		/////////////////////////////////
		E_CRYO_CTRL_STATE.WARMING_UP:
		/////////////////////////////////
		//
		// Trigger temperature ramp to in_ptr_Cryo_Ctrl^.cfg.lrTemp_Warm (~10C)
		SIM_Temp_Mirror.M_RampTo(
			in_lrValueEnd	:= in_ptr_Cryo_Ctrl^.cfg.lrTemp_Warm + 1.0,
			in_nPeriod		:= nRampPeriod);
			
			
		// Trigger temperature ramp to in_ptr_Cryo_Ctrl^.cfg.lrTemp_Warm (~10C)
		// Speed up the ramp compared to the Bench, so
		// DET temperature is slightly higher during warm-up.
		// The final temperature is the same as for the Bench.
		SIM_Temp_DET.M_RampTo(
			in_lrValueEnd	:= in_ptr_Cryo_Ctrl^.cfg.lrTemp_Warm + 1.0,
			in_nPeriod		:= nRampPeriod - 2000);
			
		/////////////////////////////////
		E_CRYO_CTRL_STATE.REPRESSURIZING:
		/////////////////////////////////
		//
		// Trigger Cryo vacuum ramp to atmospheric pressure ~820 mbar
		SIM_Pressure_Cryo.M_RampTo(
			in_lrValueEnd	:= 820.0,
			in_nPeriod		:= 17000);
			
		// Follow the same ramp with Evac but a bit slower.
		SIM_Pressure_Evac.M_RampTo(
			in_lrValueEnd	:= 820.0,
			in_nPeriod		:= 20000);
	END_CASE

END_IF


//
// Evacuation Pressure simulation
//
// Capture Evacuation ON/OFF trigger
trgEvacOn(CLK := in_ptr_Cryo_Ctrl^.ctrl.bEnable_Evac);
trgEvacOff(CLK := in_ptr_Cryo_Ctrl^.ctrl.bEnable_Evac);
IF	trgEvacOn.Q THEN
	// Trigger vacuum ramp 0.0001 mbar below Good Vacuum
	SIM_Pressure_Cryo.M_StartCurve(
		in_lrValueEnd	:= in_ptr_Cryo_Ctrl^.Pressure_Cryo.in_lrLimitGoodVac - 0.0001, 
		in_nPeriod		:= 20000, 
		in_lrCurveScale	:= 0.3);
ELSIF trgEvacOff.Q THEN
	// Evacuation stopped.
	// Keep the pressure as it is.
	SIM_Pressure_Cryo.M_Stop();
END_IF


//
// If Turbo Pump is running, keep Evacuation pressure 1.0e-05 below the Cryo pressure.
// Value is calculated on every cycle.
//
IF in_ptr_Cryo_Ctrl^.EvacSys.stat.bTurboPumpON THEN
	SIM_Pressure_Evac.M_SetValue(SIM_Pressure_Cryo.lrPress - 1.0E-05);
END_IF


//
// To get more realistic evacuation,
// Restart simulated curve when inVacuum is triggered.
//
//trgInVacuum(CLK := in_ptr_Cryo_Ctrl^.Pressure_Cryo.stat.bInVacuum);
trgInVacuum(CLK := in_ptr_Cryo_Ctrl^.stat.bInVacuum);
IF trgInVacuum.Q THEN
	SIM_Pressure_Cryo.M_StartCurve(
		in_lrValueEnd	:= in_ptr_Cryo_Ctrl^.Pressure_Cryo.in_lrLimitGoodVac - 0.0001, 
		in_nPeriod		:= 10000, 
		in_lrCurveScale	:= 0.3);
END_IF

			
//
// Capture events when buttons are released 
// and temperature transitions interrupted.
//

// Capture pre-cooling, cooling or warmup button release.
// Stop ramping in that case.
trgPrecoolOff	(CLK:=in_ptr_Cryo_Ctrl^.ctrl.bEnable_Precool);
trgCoolOff		(CLK:=in_ptr_Cryo_Ctrl^.ctrl.bEnable_Cool);
trgWarmupOff	(CLK:=in_ptr_Cryo_Ctrl^.ctrl.bEnable_Warmup);

IF	trgPrecoolOff.Q OR trgCoolOff.Q OR trgWarmupOff.Q	THEN
	SIM_Temp_Mirror.M_Stop();
	SIM_Temp_DET.M_Stop();
END_IF

END_FUNCTION_BLOCK

// POUs/System/FB_CRYO_CTRL
// Cryogenic Controller Example - ESO IRATEC
FUNCTION_BLOCK FB_CRYO_CTRL
VAR_INPUT
END_VAR
VAR

	///////////////////////////
	// Configuration parameters
	///////////////////////////
	cfg:	T_CRYO_CFG;
	
	/////////////////////
	// Control parameters
	/////////////////////
	ctrl:	T_CRYO_CTRL;

	/////////////////////
	// Status parameters
	/////////////////////
	stat:	T_CRYO_STAT;


	/////////////////////
	// System Logging
	/////////////////////
	syslog:	T_CRYO_LOG;


	/////////////////////
	// Local variables
	/////////////////////



	{attribute 'OPC.UA.DA' := '0'}
	timer:		TON;		// Timer for commands
	
	{attribute 'OPC.UA.DA' := '0'}
	ptrLog:		ARRAY [0..9] OF POINTER TO STRING(80);
	{attribute 'OPC.UA.DA' := '0'}
	nLogPos:	INT := -1;
	
	

//////////////////////////////////////////////
//             Controllers
//////////////////////////////////////////////

//
// LN2 Valve control
//
	{attribute 'OPC.UA.DA' := '1'}
	LN2: 			FB_CRYO_LN2_CTRL;
	
//
// Repressurizing Valve control
//
	{attribute 'OPC.UA.DA' := '1'}
	RepressValve:	FB_CRYO_VALVE_CTRL;
	
	
//
// Evacuation Valve control
//
	EvacSys:	FB_CRYO_EVACUATION_SYSTEM;

//
// Heater control
//
	{attribute 'OPC.UA.DA' := '1'}
	Heater: 		FB_CRYO_HEATER_CTRL;
	
//
// CCC control
//
	{attribute 'OPC.UA.DA' := '1'}
	CCC:			FB_CRYO_CCC_CTRL;

//
// CCC control
//
//	{attribute 'OPC.UA.DA' := '1'}
	Lakeshore:		FB_LAKESHORE_RS;
	
	// Compressor	
	cpa:	FB_CRYO_CPA;

//////////////////////////////////////////////
//             Sensors
//////////////////////////////////////////////
 
//
// VACUUM Sensors
//
	{attribute 'OPC.UA.DA' := '1'}
	Pressure_Cryo:		FB_CRYO_PRESSURE;	
	{attribute 'OPC.UA.DA' := '1'}
	Pressure_Evac:		FB_CRYO_PRESSURE;	
	
 
///////////////////////////////////////////////////////
//                  Temperatures
///////////////////////////////////////////////////////
 
//
// PT100 Temperatures
//
	Temp_Ambient:		FB_CRYO_TEMPERATURE;	// Ambient temperature
	Temp_ColdBench:		FB_CRYO_TEMPERATURE;	// Cold Bench temperature
	Temp_LN2_Exhaust:	FB_CRYO_TEMPERATURE;	// LN2 Exhaust temperature
	Temp_LN2_Inlet:		FB_CRYO_TEMPERATURE;	// LN2 Inlet   temperature
	Temp_Mirror:		FB_CRYO_TEMPERATURE;	// Entrance Mirror temperature
	Temp_WarmUp:		FB_CRYO_TEMPERATURE;	// Reference temperature for WarmUp

//
// Lakeshore temperatures
//
	Temp_DET:			FB_CRYO_TEMPERATURE;	// Lakeshore Channel A
	Temp_HeatShield:	FB_CRYO_TEMPERATURE;	// Heat Shield Lakeshore Channel B
 
//
// IRATEC specific Temperatures
//
	Temp_FW:			FB_CRYO_TEMPERATURE;	// Filter Wheel temperature

	

//
// System triggers
//	
	{attribute 'OPC.UA.DA' := '0'}
	trgPrecool:			R_TRIG;
	{attribute 'OPC.UA.DA' := '0'}
	trgCool:			R_TRIG;
	{attribute 'OPC.UA.DA' := '0'}
	trgWarmup:			R_TRIG;
	{attribute 'OPC.UA.DA' := '0'}
	trgRepress:			R_TRIG;
	{attribute 'OPC.UA.DA' := '0'}
	trgEvacOn:			R_TRIG;
	{attribute 'OPC.UA.DA' := '0'}
	trgEvacOff:			F_TRIG;

//
//	Input signals
//	
	i_bEvacRootPumpOK		AT%I*:	BOOL;
	i_bEvacTurboPumpOK		AT%I*:	BOOL;
	i_bEmergencySTOP		AT%I*:	BOOL;
	i_bManualOverride		AT%I*:	BOOL;
	i_bVacPumpConnected		AT%I*:	BOOL;
	i_bLN2TankConnected		AT%I*:	BOOL;
	i_bRepressLN2Connected	AT%I*:	BOOL;


//
// Dummy values for simulation, etc.
//
	// Dummy OP state for mapping of simulated devices.
	q_nStateDummy	AT%Q*:	UINT := 8;		

	
END_VAR

// Increment cycle counter
stat.nCycleCounter := stat.nCycleCounter + 1;

// Wait until the controller is configured.
IF NOT stat.bConfigured THEN
	M_Configure(); 
	RETURN;
END_IF


//
// Read Temperature and Pressure Sensors
//
M_ReadSensors();


//
// Check for sensor HW errors
//
M_CheckForSensorErrors();



///////////////////
// System Operation
///////////////////

//
// Execute Controllers
//
M_ExecuteControllers();


//
// Capture system commands
//
M_CheckForCommands();


//
// Perform a safety check
//
M_SafetyCheck();


//
// Execute system state machine
//
M_StateMachine();

METHOD M_CheckForCommands
VAR_INPUT
END_VAR
// Capture precooling command
trgPrecool(CLK := ctrl.bEnable_Precool);
IF	trgPrecool.Q AND 
	(stat.nState = E_CRYO_CTRL_STATE.WARM_VACUUM OR stat.nState = E_CRYO_CTRL_STATE.PRE_COOLED) THEN
	ctrl.bExecute	:= TRUE;
	ctrl.nCommand	:= E_CRYO_CTRL_CMD.PRECOOL;
END_IF


// Capture Cool command
trgCool(CLK := ctrl.bEnable_Cool);
IF	trgCool.Q AND stat.nState = E_CRYO_CTRL_STATE.PRE_COOLED THEN
	ctrl.bExecute	:= TRUE;
	ctrl.nCommand	:= E_CRYO_CTRL_CMD.COOL;
END_IF


// Capture Warmup command
trgWarmup(CLK := ctrl.bEnable_Warmup);
IF	trgWarmup.Q AND 
	(stat.nState = E_CRYO_CTRL_STATE.PRE_COOLED OR stat.nState = E_CRYO_CTRL_STATE.COLD) THEN
	ctrl.bExecute	:= TRUE;
	ctrl.nCommand	:= E_CRYO_CTRL_CMD.WARM_UP;
END_IF


// Capture Repressure command
trgRepress(CLK := ctrl.bEnable_RepressCtrl);
IF	trgRepress.Q AND 
	(stat.nState = E_CRYO_CTRL_STATE.WARM_VACUUM) THEN
	ctrl.bExecute	:= TRUE;
	ctrl.nCommand	:= E_CRYO_CTRL_CMD.REPRESSURIZE;
END_IF


// Capture Evacuation ON/OFF trigger
trgEvacOn(CLK := ctrl.bEnable_Evac);
trgEvacOff(CLK := ctrl.bEnable_Evac);
IF	trgEvacOn.Q AND NOT ctrl.bEnable_RepressSys THEN
	ctrl.bEnable_Evac	:= TRUE;
	M_SysLog('Evacuation started.');
ELSIF trgEvacOff.Q THEN
	ctrl.bEnable_Evac	:= FALSE;
	M_SysLog('Evacuation stopped.');
END_IF
END_METHOD

METHOD M_CheckForSensorErrors
VAR_INPUT
END_VAR
////////////////////////////////////////////////
// Check for errors by testing the 'Valid' flag.
////////////////////////////////////////////////
IF		NOT Pressure_Cryo.stat.bValid	THEN
	stat.bError	:= TRUE;
	stat.sState	:= 'Cryo Vacuum gauge problem';
	stat.nState	:= E_CRYO_CTRL_STATE.ERROR;
ELSIF	NOT Temp_Mirror.stat.bValid	THEN
	stat.bError	:= TRUE;
	stat.sState	:= 'Mirror Temperature sensor problem';
	stat.nState	:= E_CRYO_CTRL_STATE.ERROR;
ELSE
	stat.bError	:= FALSE;
	stat.sState	:= '';
END_IF


///////////////////////
// Check for Interlocks
///////////////////////

//
// Evacuation and Repressurization are mutually exclusive.
//
IF EvacSys.in_bEnable THEN
	ctrl.bEnable_RepressSys	:= FALSE;
ELSIF RepressValve.in_bEnable THEN
	ctrl.bEnable_Evac	:= FALSE;
END_IF

//
// Disable control in failure state
//
IF stat.bError THEN
	ctrl.bEnable_Precool	:= FALSE;
	ctrl.bEnable_Cool 		:= FALSE;
	ctrl.bEnable_Warmup		:= FALSE;
END_IF
END_METHOD

METHOD M_CheckLakeshoreCommand
VAR_INPUT
END_VAR
(* TODO

IF ctrl.bLS_UpdateSETP THEN
	// Reset trigger flag
	ctrl.bLS_UpdateSETP	:= FALSE;
	
	// Safety
	IF ctrl.lrLS_RAMP > 1.0 THEN
		ctrl.lrLS_RAMP	:= 1.0;
	ELSIF ctrl.lrLS_RAMP < 0.0 THEN
		ctrl.lrLS_RAMP	:= 0.0;
	END_IF
	
	// Set the mode
	IF ctrl.nLS_Mode <> E_CRYO_LAKESHORE_MODE.MONITORING THEN
		Lakeshore.M_SetMode(ctrl.nLS_Mode);
	ELSE
		RETURN;	// Nothing to do
	END_IF
ELSE
	RETURN;	// Nothing to do
END_IF




CASE ctrl.nLS_Mode OF
	E_CRYO_LAKESHORE_MODE.MONITORING,
	E_CRYO_LAKESHORE_MODE.COOLING,
	E_CRYO_LAKESHORE_MODE.WARMUP,
	E_CRYO_LAKESHORE_MODE.COOLING_UPDATE,
	E_CRYO_LAKESHORE_MODE.WARMUP_UPDATE:
		Lakeshore.M_SetMode(E_CRYO_LAKESHORE_MODE.MONITORING);	// No action
		
	E_CRYO_LAKESHORE_MODE.SINGLE_SETUP:
		IF stat.nState = E_CRYO_CTRL_STATE.COLD THEN
			Lakeshore.M_SetParams(
				in_nPID_A_P			:= cfg.LS_W_PID_A_P, 
				in_nPID_A_I			:= cfg.LS_W_PID_A_I, 
				in_nPID_A_D			:= cfg.LS_W_PID_A_D, 
				in_nHeater_Range	:= cfg.LS_W_Heater_Range, 
				in_lrCtrlRamp		:= ctrl.lrLS_RAMP, 
				in_lrSetpoint_A		:= ctrl.lrLS_SETP);
		END_IF
	ELSE
		Lakeshore.M_SetMode(E_CRYO_LAKESHORE_MODE.MONITORING);	// No action
END_CASE
*)
END_METHOD

// Method to check status of the cryostat vacuum.
// TODO: The limits might depend on the temperature.
METHOD M_CheckVacuum
VAR_INPUT
END_VAR
IF Pressure_Cryo.stat.bValid  THEN
	IF Pressure_Cryo.stat.lrPressure < cfg.lrPress_GoodVac THEN
		stat.bInVacuum	:= TRUE;
		stat.bGoodVacuum:= TRUE;
	ELSIF Pressure_Cryo.stat.lrPressure < cfg.lrPress_InVac THEN
		stat.bInVacuum	:= TRUE;
		stat.bGoodVacuum:= FALSE;
	ELSE
		stat.bInVacuum	:= FALSE;
		stat.bGoodVacuum:= FALSE;
	END_IF 
ELSE
	stat.bInVacuum	:= FALSE;
	stat.bGoodVacuum:= FALSE;
END_IF
END_METHOD

METHOD M_Configure
VAR_INPUT
END_VAR
IF stat.bConfigured THEN
	RETURN;
ELSIF stat.nCycleCounter = 100 THEN
	// Set pointers to system logs.
	ptrLog[0] := ADR(syslog.s0);
	ptrLog[1] := ADR(syslog.s1);
	ptrLog[2] := ADR(syslog.s2);
	ptrLog[3] := ADR(syslog.s3);
	ptrLog[4] := ADR(syslog.s4);
	ptrLog[5] := ADR(syslog.s5);
	ptrLog[6] := ADR(syslog.s6);
	ptrLog[7] := ADR(syslog.s7);
	ptrLog[8] := ADR(syslog.s8);
	ptrLog[9] := ADR(syslog.s9);
ELSIF stat.nCycleCounter > 200 THEN
	stat.bConfigured	:= TRUE;
ELSE
	RETURN;
END_IF
END_METHOD

METHOD M_ExecuteControllers
VAR
END_VAR
//
// Controllers, i.e. LN2 cooler, Heater, ...
//

// Activate Lakeshore SETP command, if any (see ctrl.xxLS_...)
M_CheckLakeshoreCommand();

// Execute Lakeshore 340 controller
Lakeshore(
	in_bSimulation	:= TRUE,
	in_sName		:= 'LS340',
	in_nModel		:= 340, 
	in_bAutoMonitor	:= TRUE, 
	in_nPeriod 		:= 2000,
	in_sCmdSuffix	:= '$0D$0A',
	in_sReplySuffix	:= '$0D$0A');


LN2(
	in_bEnable			:= ctrl.bEnable_Precool, 
	in_nFeedback		:= E_CRYO_BIN_ACT_FEEDBACK.ON_ONLY, 
	in_lrTempK			:= Temp_LN2_Exhaust.stat.lrTempK, 
	in_bValid			:= Temp_LN2_Exhaust.stat.bValid, 
	in_lrTempValveOpen	:= cfg.lrTemp_LN2ValveOpen, 
	in_lrTempValveClose	:= cfg.lrTemp_LN2ValveClose);
	
RepressValve(in_bEnable	:= ctrl.bEnable_RepressCtrl);
	
EvacSys(
	in_bEnable			:= ctrl.bEnable_Evac,
	in_Pressure_Cryo	:= Pressure_Cryo.stat,
	in_Pressure_Evac	:= Pressure_Evac.stat,
	in_Temp_Cryo		:= Temp_Mirror.stat,
	in_bRepressValveOpen:= RepressValve.stat.bActON, 
	in_bRepressValveOK	:= NOT RepressValve.stat.bError);

	
// Heater compares DET temperature against the lowest temperature in the system. 
// Lowest temperature is calculated in M_ReadSensors() by 
// calling M_GetLowestTemperature().
Heater(
	in_bEnable		:= (ctrl.bEnable_Heater AND NOT i_bEmergencySTOP), 
	in_nFeedback	:= E_CRYO_BIN_ACT_FEEDBACK.ON_ONLY, 
	in_lrTemp1		:= stat.lrHighestTempK, 
	in_lrTemp2		:= Temp_DET.stat.lrTempK, 
	in_bValidTemp1	:= stat.bHighestTempValid,
	in_bValidTemp2	:= Temp_DET.stat.bValid,
	in_lrDelta_Low	:= cfg.lrTemp_DeltaDet_Bench_Low, 
	in_lrDelta_High	:= cfg.lrTemp_DeltaDet_Bench_High);

	
CCC(in_bEnable	:= ctrl.bEnable_CCC);


cpa(in_bSimulation				:= FALSE,
	in_sName					:= 'PT810-01',
	in_sSN_Compressor			:= 'CPA289C-W2EHCE-180201A',
	in_sSN_PulseTube			:= 'CH40810-180208A',
	in_nYear_Compressor			:= 2018,
	in_nYear_PulseTube			:= 2020,
	in_lrNextService_Compressor	:= 20000.0,
	in_lrNextService_PulseTube	:= 35000.0,
	in_nSlaveID					:= 16,
	in_nPeriod					:= 1000);
END_METHOD

METHOD M_GetHighestTemperature
VAR_INPUT
END_VAR
VAR
	lrTempK:	LREAL	:= 0.0;	// The lowest possible temperature
	bValid:		BOOL	:= FALSE;
END_VAR
//
// Get the warmest temperature among Mirror, Bench, FilterWheel and WarmUp
//

// If there is at least one Valid reading, the result is valid.
IF	Temp_Mirror.stat.bValid 	OR 
	Temp_ColdBench.stat.bValid	OR 
	Temp_FW.stat.bValid			OR 
	Temp_WarmUp.stat.bValid			THEN
	bValid	:= TRUE;
END_IF


// Get the highest temperature from Valid temperatures.
// Take Mirror temperature first, if Valid.
// If not Valid, try with WarmUp sensor.
// If that doesn't work, take the Filter Wheel temperature.
IF Temp_Mirror.stat.bValid THEN
	IF Temp_Mirror.stat.lrTempK > lrTempK THEN
		lrTempK	:= Temp_Mirror.stat.lrTempK;
	END_IF
ELSIF Temp_WarmUp.stat.bValid THEN
	IF Temp_WarmUp.stat.lrTempK > lrTempK THEN
		lrTempK	:= Temp_Mirror.stat.lrTempK;
	END_IF
ELSIF Temp_FW.stat.bValid THEN
	IF Temp_FW.stat.lrTempK > lrTempK THEN
		lrTempK	:= Temp_Mirror.stat.lrTempK;
	END_IF
END_IF


// Update status
stat.lrHighestTempK		:= lrTempK;
stat.bHighestTempValid	:= bValid;
END_METHOD

METHOD M_GetLowestTemperature
VAR_INPUT
END_VAR
VAR
	lrTempK:	LREAL	:= 293.15;	// Room temperature 20 C
	bValid:		BOOL	:= FALSE;
END_VAR
//
// Get the coldest temperature among Mirror, Bench, FilterWheel and WarmUp
//

// If there is at least one Valid reading, the result is valid.
IF	Temp_Mirror.stat.bValid 	OR 
	Temp_ColdBench.stat.bValid	OR 
	Temp_FW.stat.bValid			OR 
	Temp_WarmUp.stat.bValid			THEN
	bValid	:= TRUE;
END_IF


// Get the lowest temperature from Valid temperatures.
IF Temp_Mirror.stat.bValid AND Temp_Mirror.stat.lrTempK < lrTempK THEN
	lrTempK	:= Temp_Mirror.stat.lrTempK;
END_IF

IF Temp_ColdBench.stat.bValid AND Temp_ColdBench.stat.lrTempK < lrTempK THEN
	lrTempK	:= Temp_ColdBench.stat.lrTempK;
END_IF

IF Temp_FW.stat.bValid AND Temp_FW.stat.lrTempK < lrTempK THEN
	lrTempK	:= Temp_FW.stat.lrTempK;
END_IF

IF Temp_WarmUp.stat.bValid AND Temp_WarmUp.stat.lrTempK < lrTempK THEN
	lrTempK	:= Temp_WarmUp.stat.lrTempK;
END_IF

// Update status
stat.lrLowestTempK		:= lrTempK;
stat.bLowestTempValid	:= bValid;

// Get Temperature difference (DET -Lowest temperature) [K]
IF stat.bLowestTempValid  AND  Temp_DET.stat.bValid  THEN
	stat.bDiffTempValid	:= TRUE;
	stat.lrDiffTempK	:= Temp_DET.stat.lrTempK - stat.lrLowestTempK;
ELSE
	stat.bDiffTempValid	:= FALSE;
	stat.lrDiffTempK	:= -100;
END_IF
END_METHOD

METHOD M_GetState
VAR_INPUT
END_VAR
// Determine the initial state based on the command and actuator state.
IF NOT stat.bCtrlOK	THEN
	stat.nState	:= E_CRYO_CTRL_STATE.ERROR;
ELSIF	Temp_Mirror.stat.lrTempK >= cfg.lrTemp_Precooled  AND  NOT stat.bInVacuum	THEN
	stat.nState	:= E_CRYO_CTRL_STATE.WARM_PRESS;
ELSIF	Temp_Mirror.stat.lrTempK >= cfg.lrTemp_Precooled  AND  stat.bInVacuum  THEN
	stat.nState	:= E_CRYO_CTRL_STATE.WARM_VACUUM;
ELSIF	Temp_Mirror.stat.lrTempK < cfg.lrTemp_Cold 	AND  stat.bInVacuum  THEN
	stat.nState	:= E_CRYO_CTRL_STATE.COLD;
ELSIF	Temp_Mirror.stat.lrTempK < cfg.lrTemp_Precooled  AND  stat.bInVacuum  THEN
	stat.nState	:= E_CRYO_CTRL_STATE.PRE_COOLED;
END_IF
M_SetStatus(stat.nState);
END_METHOD

METHOD M_ReadSensors
VAR_INPUT
END_VAR
//
// Read system temperatures, i.e. LN2, Bench and Detector temperatures
//
Temp_Ambient		(in_lrScale_1:=0.1);
Temp_ColdBench 		(in_lrScale_1:=0.1, in_bIgnoreUnderrange_1 := ctrl.bIgnoreUnderrange_ColdBench);
Temp_LN2_Exhaust	(in_lrScale_1:=0.1);
Temp_LN2_Inlet		(in_lrScale_1:=0.1);
Temp_Mirror			(in_lrScale_1:=0.1);
Temp_WarmUp			(in_lrScale_1:=0.1);

Temp_FW				(in_lrScale_1:=0.1);	// IRATEC specific

//
// Lakeshore temperature
//
// Important note:
// In normal operation, call to Temp_DET() will result in a reading that is
// not valid since the underlying temperature sensors should not be 
// mapped to temperature signals.
// However, call to Temp_DET.M_GetTemperatureFromLakeshore() will copy 
// the Lakeshore reading to it and update the Valid flag.
//
// DET temperature is Lakeshore Channel A

(* TODO
Temp_DET(in_lrScale_1:=0.1);	
Temp_DET.M_GetTemperatureFromLakeshore(
	bValid	:= (Lakeshore.stat.nErrorCode=0),
	lrTempK	:=  Lakeshore.stat.lrKRDG_A,
	lrTempC	:=  Lakeshore.stat.lrCRDG_A);

// HeatShield temperature is Lakeshore Channel B
Temp_HeatShield(in_lrScale_1:=0.1);
Temp_HeatShield.M_GetTemperatureFromLakeshore(
	bValid	:= (Lakeshore.stat.nErrorCode=0),
	lrTempK	:=  Lakeshore.stat.lrKRDG_B,
	lrTempC	:=  Lakeshore.stat.lrCRDG_B);

*)

// Both pressure sensors are of PKR250/251 type
Pressure_Cryo(	in_lrLimitInVac		:= cfg.lrPress_InVac, 
				in_lrLimitGoodVac	:= cfg.lrPress_GoodVac);
Pressure_Evac(	in_lrLimitInVac		:= cfg.lrPress_InVac, 
				in_lrLimitGoodVac	:= cfg.lrPress_GoodVac);	

//
// Get the lowest temperature in the cryostat
//	
M_GetLowestTemperature();

//
// Get the highest temperature in the cryostat
//	
M_GetHighestTemperature();
	

//
// Check Vacuum in the system
//	
M_CheckVacuum();
END_METHOD

METHOD M_SafetyCheck
VAR_INPUT
END_VAR
//
// Repressurization safety
//
IF	NOT ctrl.bEnable_Evac AND
	(stat.nState = E_CRYO_CTRL_STATE.WARM_PRESS 		OR 
	 stat.nState = E_CRYO_CTRL_STATE.REPRESSURIZING 	OR 
	 stat.nState = E_CRYO_CTRL_STATE.WARM_VACUUM) 		THEN
	ctrl.bSafe_Repress	:= TRUE;
ELSE
	ctrl.bSafe_Repress	:= FALSE;
	ctrl.bEnable_RepressSys:= FALSE;
END_IF
END_METHOD

METHOD M_SetStatus
VAR_INPUT
	nState:	E_CRYO_CTRL_STATE;
END_VAR

CASE nState OF
	
	E_CRYO_CTRL_STATE.NONE:
	stat.bDone	:= TRUE;
	stat.bBusy	:= FALSE;
	stat.bError	:= FALSE;
	stat.bActive:= FALSE;
	stat.sState	:= 'OFF';
	
	E_CRYO_CTRL_STATE.WARM_PRESS:
	stat.bDone	:= TRUE;
	stat.bBusy	:= FALSE;
	stat.bError	:= FALSE;
	stat.bActive:= TRUE;
	stat.sState	:= 'WARM  -  PRESSURIZED';
	
	E_CRYO_CTRL_STATE.WARM_VACUUM:
	stat.bDone	:= TRUE;
	stat.bBusy	:= FALSE;
	stat.bError	:= FALSE;
	stat.bActive:= TRUE;
	stat.sState	:= 'WARM  -  VACUUM';
	
	E_CRYO_CTRL_STATE.PRE_COOLING:
	stat.bDone	:= FALSE;
	stat.bBusy	:= TRUE;
	stat.bError	:= FALSE;
	stat.bActive:= TRUE;
	stat.sState	:= 'PRE-COOLING...';
	
	E_CRYO_CTRL_STATE.PRE_COOLED:
	stat.bDone	:= TRUE;
	stat.bBusy	:= FALSE;
	stat.bError	:= FALSE;
	stat.bActive:= TRUE;
	stat.sState	:= 'PRE-COOLED';

	E_CRYO_CTRL_STATE.COOLING_DOWN:
	stat.bDone	:= FALSE;
	stat.bBusy	:= TRUE;
	stat.bError	:= FALSE;
	stat.bActive:= TRUE;
	stat.sState	:= 'COOLING DOWN...';

	E_CRYO_CTRL_STATE.COLD:
	stat.bDone	:= TRUE;
	stat.bBusy	:= FALSE;
	stat.bError	:= FALSE;
	stat.bActive:= TRUE;
	stat.sState	:= 'COLD';

	E_CRYO_CTRL_STATE.WARMING_UP:
	stat.bDone	:= FALSE;
	stat.bBusy	:= TRUE;
	stat.bError	:= FALSE;
	stat.bActive	:= TRUE;
	IF Temp_Mirror.stat.lrTempK >= cfg.lrTemp_Warm	THEN
		stat.sState	:= 'WARM';
	ELSIF	Temp_Mirror.stat.lrTempK < cfg.lrTemp_Warm AND
			Temp_Mirror.stat.lrTempK >= cfg.lrTemp_Precooled	THEN
		stat.sState	:= 'WARMING UP... PRE-COOLED';
	ELSE
		stat.sState	:= 'WARMING UP... COLD';
	END_IF

	E_CRYO_CTRL_STATE.REPRESSURIZING:
	stat.bDone	:= FALSE;
	stat.bBusy	:= TRUE;
	stat.bError	:= FALSE;
	stat.bActive:= TRUE;
	stat.sState	:= 'RE-PRESSURIZING...';
	
	E_CRYO_CTRL_STATE.ERROR:
	stat.bDone	:= TRUE;
	stat.bBusy	:= FALSE;
	stat.bError	:= TRUE;
	stat.bActive:= FALSE;
	stat.sState	:= 'ERROR';

END_CASE
END_METHOD

METHOD M_StateMachine
VAR_INPUT
END_VAR
////////////////
// State Machine
////////////////
CASE stat.nState OF
	/////////////////////////////////
	E_CRYO_CTRL_STATE.NONE:
	/////////////////////////////////
	//
	// This is the state on power-up.
	// Determine the initial state based on the command and actuator state.
	M_GetState();	
	RETURN;
	

	/////////////////////////////////
	E_CRYO_CTRL_STATE.WARM_PRESS:
	/////////////////////////////////
	//
	ctrl.bSafe_Precool	:= FALSE;
	ctrl.bSafe_Cooling	:= FALSE;
	ctrl.bSafe_Warmup	:= FALSE;

	ctrl.bEnable_RepressCtrl:= FALSE;
	ctrl.bEnable_Heater		:= FALSE;

	IF	ctrl.bExecute	THEN
		ctrl.bExecute		:= FALSE;
		stat.nLastCommand	:= ctrl.nCommand;
		ctrl.nCommand		:= E_CRYO_CTRL_CMD.NONE;
	ELSIF Pressure_Cryo.stat.lrPressure < cfg.lrPress_InVac THEN
		// Evacuation is not part of the State Machine.
		// Once the air has been evacuated, we switch to WARM_VACUUM.
		stat.nState := E_CRYO_CTRL_STATE.WARM_VACUUM;
	END_IF
	M_SetStatus(stat.nState);	
	RETURN;
	
	
	//////////////////////////////////////////
	E_CRYO_CTRL_STATE.WARM_VACUUM:
	//////////////////////////////////////////
	//
	ctrl.bSafe_Precool	:= NOT ctrl.bEnable_RepressSys;
	ctrl.bSafe_Cooling	:= FALSE;
	ctrl.bSafe_Warmup	:= FALSE;
	
	// In this state CCC should be OFF
	ctrl.bEnable_CCC	:= FALSE;
	ctrl.bEnable_Heater	:= FALSE;

	IF	ctrl.bExecute	THEN
		ctrl.bExecute		:= FALSE;
		stat.nLastCommand	:= ctrl.nCommand;
		ctrl.nCommand		:= E_CRYO_CTRL_CMD.NONE;
		IF stat.nLastCommand = E_CRYO_CTRL_CMD.PRECOOL	THEN
			IF CCC.stat.bActive THEN
				ctrl.bEnable_Precool	:= FALSE;
				M_SysLog('Cannot start pre-cooling. CCC still active!');
				RETURN;
			ELSIF CCC.stat.bError THEN
				ctrl.bEnable_Precool	:= FALSE;
				M_SysLog('Cannot start pre-cooling. CCC in Error state!');
				RETURN;
			END_IF
			
			// Configure Lakeshore for Cooling
			Lakeshore.M_RampEnable(
				in_nPID_A_P			:= cfg.LS_C_PID_A_P, 
				in_nPID_A_I			:= cfg.LS_C_PID_A_I, 
				in_nPID_A_D			:= cfg.LS_C_PID_A_D, 
				in_nHeater_Range	:= cfg.LS_C_Heater_Range, 
				in_lrCtrlRamp		:= cfg.LS_C_CTRL_RAMP, 
				in_lrSetpoint_A		:= cfg.LS_C_SETPOINT_A);
			
			M_SysLog('Pre-cooling started.');
			stat.nState	:= E_CRYO_CTRL_STATE.PRE_COOLING;
		ELSIF stat.nLastCommand = E_CRYO_CTRL_CMD.REPRESSURIZE	THEN
			// Disable Evacuation Valve control
			ctrl.bEnable_Evac	:= FALSE;
			ctrl.bEnable_RepressCtrl := TRUE;
			
			// Configure Lakeshore just to monitor. Disable control.
			Lakeshore.M_RampDisable();

			M_SysLog('Re-pressurization started.');
			stat.nState	:= E_CRYO_CTRL_STATE.REPRESSURIZING;
		END_IF
	END_IF
	M_SetStatus(stat.nState);	
	RETURN;
	

	/////////////////////////////////
	E_CRYO_CTRL_STATE.PRE_COOLING:
	/////////////////////////////////
	//
	ctrl.bSafe_Precool	:= TRUE;
	ctrl.bSafe_Cooling	:= FALSE;
	ctrl.bSafe_Warmup	:= FALSE;

	ctrl.bEnable_CCC	:= FALSE;

	ctrl.bEnable_RepressCtrl:= FALSE;

	IF Temp_Mirror.stat.lrTempK < cfg.lrTemp_Precooled	THEN
		M_SysLog('Pre-cooling complete. State is Pre-cooled.');
		stat.nState	:= E_CRYO_CTRL_STATE.PRE_COOLED;
	ELSIF NOT ctrl.bEnable_Precool THEN
		// Pre-cooling has been interrupted.
		// Go back to WARM_VACUUM state.
		M_SysLog('Pre-cooling interrupted. State is Warm-Vacuum.');
		stat.nState := E_CRYO_CTRL_STATE.WARM_VACUUM;
	END_IF
	M_SetStatus(stat.nState);	
	RETURN;
	
	
	///////////////////////////////////////////
	E_CRYO_CTRL_STATE.PRE_COOLED:
	///////////////////////////////////////////
	//
	ctrl.bSafe_Precool	:= TRUE;
	ctrl.bSafe_Cooling	:= NOT ctrl.bEnable_Precool;
	ctrl.bSafe_Warmup	:= NOT ctrl.bEnable_Precool;
	ctrl.bEnable_CCC	:= FALSE;

	ctrl.bEnable_RepressCtrl:= FALSE;

	//
	// Only COOL and WARM_UP commands are allowed in state PRE_COOLED.
	// Other commands are ignored.
	//
	IF	ctrl.bExecute	THEN
		ctrl.bExecute		:= FALSE;
		stat.nLastCommand	:= ctrl.nCommand;
		ctrl.nCommand		:= E_CRYO_CTRL_CMD.NONE;
		IF stat.nLastCommand = E_CRYO_CTRL_CMD.COOL	THEN
			IF LN2.stat.bActive THEN
				M_SysLog('Cannot start cooling. LN2 still active!');
				RETURN;
			ELSIF LN2.stat.bError THEN
				M_SysLog('Cannot start cooling. LN2 in Error state!');
				RETURN;
			END_IF

			// Configure Lakeshore for cooling
			Lakeshore.M_RampEnable(
				in_nPID_A_P			:= cfg.LS_C_PID_A_P, 
				in_nPID_A_I			:= cfg.LS_C_PID_A_I, 
				in_nPID_A_D			:= cfg.LS_C_PID_A_D, 
				in_nHeater_Range	:= cfg.LS_C_Heater_Range, 
				in_lrCtrlRamp		:= cfg.LS_C_CTRL_RAMP, 
				in_lrSetpoint_A		:= cfg.LS_C_SETPOINT_A);
			
			M_SysLog('Cool-down started.');
			stat.nState	:= E_CRYO_CTRL_STATE.COOLING_DOWN;
		ELSIF stat.nLastCommand = E_CRYO_CTRL_CMD.WARM_UP	THEN
			// Eable Evacuation Valve control here.
			// This way the user will be able to turn it on/off
			// during the warmup phase.
			ctrl.bEnable_Evac	:= TRUE;

			// Configure Lakeshore for Warmup
			Lakeshore.M_RampEnable(
				in_nPID_A_P			:= cfg.LS_W_PID_A_P, 
				in_nPID_A_I			:= cfg.LS_W_PID_A_I, 
				in_nPID_A_D			:= cfg.LS_W_PID_A_D, 
				in_nHeater_Range	:= cfg.LS_W_Heater_Range, 
				in_lrCtrlRamp		:= cfg.LS_W_CTRL_RAMP, 
				in_lrSetpoint_A		:= cfg.LS_W_SETPOINT_A);
			
			M_SysLog('Warm-up started.');
			stat.nState	:= E_CRYO_CTRL_STATE.WARMING_UP;
		END_IF
	END_IF
	M_SetStatus(stat.nState);	
	RETURN;
	
	/////////////////////////////////
	E_CRYO_CTRL_STATE.COOLING_DOWN:
	/////////////////////////////////
	//
	ctrl.bSafe_Precool	:= FALSE;
	ctrl.bSafe_Cooling	:= TRUE;
	ctrl.bSafe_Warmup	:= FALSE;
	ctrl.bEnable_CCC	:= TRUE;

	ctrl.bEnable_RepressCtrl:= FALSE;
	
	IF Temp_Mirror.stat.lrTempK < cfg.lrTemp_Cold	THEN
		M_SysLog('Cool-down complete. State is Cold.');
		// Enable Evacuation Valve control
		ctrl.bEnable_Evac	:= TRUE;
		stat.nState	:= E_CRYO_CTRL_STATE.COLD;
	ELSIF NOT ctrl.bEnable_Cool THEN
		// Cooling has been interrupted.
		// Go back to PRE_COOLED state.
		M_SysLog('Cooling interrupted. State is Pre-cooled.');
		stat.nState := E_CRYO_CTRL_STATE.PRE_COOLED;
	END_IF
	M_SetStatus(stat.nState);	
	RETURN;
	
	
	///////////////////////////////////////////
	E_CRYO_CTRL_STATE.COLD:
	///////////////////////////////////////////
	//
	ctrl.bSafe_Precool	:= FALSE;
	ctrl.bSafe_Cooling	:= TRUE;
	ctrl.bSafe_Warmup	:= NOT ctrl.bEnable_Cool;

	ctrl.bEnable_CCC		:= TRUE;
	ctrl.bEnable_RepressCtrl:= FALSE;

	//
	// Only WARM_UP command is allowed in state COLD.
	// Other commands are ignored.
	//
	IF	ctrl.bExecute	THEN
		ctrl.bExecute		:= FALSE;
		stat.nLastCommand	:= ctrl.nCommand;
		ctrl.nCommand		:= E_CRYO_CTRL_CMD.NONE;
		IF stat.nLastCommand = E_CRYO_CTRL_CMD.WARM_UP	THEN
			// Turbo OK
			// CCC OFF - by Hand (button)
			// LN2 OFF
			
			// Eable Evacuation Valve control here.
			// This way the user will be able to turn it on/off
			// during the warmup phase.
			ctrl.bEnable_Evac	:= TRUE;

			// Configure Lakeshore for Warmup
			Lakeshore.M_RampEnable(
				in_nPID_A_P			:= cfg.LS_W_PID_A_P, 
				in_nPID_A_I			:= cfg.LS_W_PID_A_I, 
				in_nPID_A_D			:= cfg.LS_W_PID_A_D, 
				in_nHeater_Range	:= cfg.LS_W_Heater_Range, 
				in_lrCtrlRamp		:= cfg.LS_W_CTRL_RAMP, 
				in_lrSetpoint_A		:= cfg.LS_W_SETPOINT_A);
			
			M_SysLog('Warm-up started.');
			stat.nState	:= E_CRYO_CTRL_STATE.WARMING_UP;
		END_IF
	END_IF
	M_SetStatus(stat.nState);	
	RETURN;
	
	/////////////////////////////////
	E_CRYO_CTRL_STATE.WARMING_UP:
	/////////////////////////////////
	//
	ctrl.bSafe_Precool	:= FALSE;
	ctrl.bSafe_Cooling	:= FALSE;

	ctrl.bEnable_Heater := TRUE;

	// In this state CCC should be OFF
	ctrl.bEnable_CCC	:= FALSE;
	
	// Switch LN2 OFF
	ctrl.bEnable_Precool	:= FALSE;
	
	// Block re-pressurisation subsystem
	ctrl.bEnable_RepressCtrl:= FALSE;

	// TODO: ???
	// Evac.stat.bActON must be all the time. 
	// If not, error AND 
	// ctrl.bEnable_Heater := false; AND
	// Re-configure Lakeshore for IDLE (no warming)

	IF Temp_Mirror.stat.lrTempK > cfg.lrTemp_Warm	THEN
		// Cryo temperature is higher than the Warm threshold.
		// The cryo is in WARM_VACUUM state.
		ctrl.bEnable_Warmup	:= FALSE;
		M_SysLog('Warm-up complete. State is Warm-Vacuum.');
		stat.nState	:= E_CRYO_CTRL_STATE.WARM_VACUUM;
	ELSIF NOT ctrl.bEnable_Warmup THEN
		// Warming up has been interrupted.
		// Based on the Bench temperature determine whether
		// the Cryo is in PRE_COOLED or COLD state.
		IF	Temp_Mirror.stat.lrTempK <  cfg.lrTemp_Warm AND
			Temp_Mirror.stat.lrTempK >= cfg.lrTemp_Precooled	THEN
			// Go back to PRE_COOLED state.
			M_SysLog('Warming up interrupted. State is Pre-cooled.');
			stat.nState := E_CRYO_CTRL_STATE.PRE_COOLED;
		ELSE
			// Go back to COLD state.
			M_SysLog('Warming up interrupted. State is Cold.');
			stat.nState := E_CRYO_CTRL_STATE.COLD;
		END_IF
	END_IF
	M_SetStatus(stat.nState);	
	RETURN;
	
	
	/////////////////////////////////
	E_CRYO_CTRL_STATE.REPRESSURIZING:
	/////////////////////////////////
	//
	ctrl.bSafe_Precool	:= FALSE;
	ctrl.bSafe_Cooling	:= FALSE;
	ctrl.bSafe_Warmup	:= FALSE;

	ctrl.bEnable_CCC	:= FALSE;

	IF	Temp_Mirror.stat.lrTempK > cfg.lrTemp_Precooled	AND  
		Pressure_Cryo.stat.lrPressure >= cfg.lrPress_Atm  		THEN
		ctrl.bEnable_RepressCtrl	:= FALSE;
		// Disable Evacuation Valve control
		ctrl.bEnable_Evac	:= FALSE;
		M_SysLog('Re-pressurization complete. State is Warm-Pressurized.');
		stat.nState	:= E_CRYO_CTRL_STATE.WARM_PRESS;
	ELSIF NOT ctrl.bEnable_RepressCtrl THEN
		// Re-pressurization has been interrupted.
		// Go back to WARM_VACUUM state.
		M_SysLog('Re-pressurization interrupted. State is Warm-Vacuum.');
		stat.nState := E_CRYO_CTRL_STATE.WARM_VACUUM;
	END_IF
	M_SetStatus(stat.nState);	
	RETURN;
	
	
	/////////////////////////////////
	E_CRYO_CTRL_STATE.ERROR:
	/////////////////////////////////
	//
	// RESET the controller in order to try to clear error
	IF ctrl.bReset THEN
		ctrl.bReset	:= FALSE;	// Clear RESET flag
		// Goto NONE state
		stat.nState	:= E_CRYO_CTRL_STATE.NONE;
		M_SetStatus(stat.nState);	
	ELSIF NOT stat.bError  THEN
		// Goto NONE state
		stat.nState	:= E_CRYO_CTRL_STATE.NONE;
		M_SetStatus(stat.nState);	
	END_IF
	RETURN;

END_CASE
END_METHOD

METHOD M_SysLog
VAR_INPUT
	str:	STRING(80);
END_VAR
VAR
	i:	INT;
END_VAR
nLogPos	:= nLogPos + 1;
IF nLogPos > 9 THEN
	FOR i := 1 TO 9 DO
		// Shift last 9 readings
		ptrLog[i-1]^ := ptrLog[i]^;
	END_FOR
	nLogPos	:= 9;
END_IF

ptrLog[nLogPos]^ := str;
END_METHOD

END_FUNCTION_BLOCK

// POUs/Subsystems/Evacuation/FB_CRYO_EVACUATION_SYSTEM
//
// Evacuation System Controller.
// The system consists of:
// - Evacuation Valve
// - Root Pump
// - Turbo Pump
//
FUNCTION_BLOCK FB_CRYO_EVACUATION_SYSTEM
VAR_INPUT
	in_Cryo_Cfg:			T_CRYO_CFG;					// Cryo configuration
	in_Temp_Cryo:			T_CRYO_TEMPERATURE_STATUS;	// Cold Bench temperature	
	in_Pressure_Cryo:		T_CRYO_PRESSURE_STATUS;		// Cryostat Pressure
	in_Pressure_Evac:		T_CRYO_PRESSURE_STATUS;		// Evacuation Pressure
	
	in_bRepressValveOpen:	BOOL;	// Repressure Valve Open flag
	in_bRepressValveOK:		BOOL;	// Repressure Valve OK flag
	in_nFeedback:	E_CRYO_BIN_ACT_FEEDBACK := E_CRYO_BIN_ACT_FEEDBACK.ON_ONLY;	// Feedbacks
	// Time between closing Vac valve and Switching OFF the vac Pump [ms]
	in_nTimeout:	UDINT := 3200;	// Timeout for switching on/off [ms]
	in_bEnable:		BOOL := FALSE;	// Controller active while in_bEnable is TRUE
	in_bCmd:		BOOL := FALSE;	// ON=TRUE, OFF=FALSE
END_VAR
VAR
	
	{attribute 'OPC.UA.DA' := '0'}
	i_bRootPumpOn	AT%I*:	BOOL;		// Root Pump Feedback
	{attribute 'OPC.UA.DA' := '0'}
	i_bTurboPumpOn	AT%I*:	BOOL;		// Turbo Pump Feedback
	
	{attribute 'OPC.UA.DA' := '0'}
	q_bPumpCtrl		AT%Q*:	BOOL;			// Pump Control signal
	
	stat:			T_CRYO_EVACUATION_SYSTEM_STATUS;

	{attribute 'OPC.UA.DA' := '1'}
	Valve:	FB_CRYO_BIN_ACT;			// Evacuation Valve 

	{attribute 'OPC.UA.DA' := '0'}
	bExecute_Valve:	BOOL := FALSE;

	{attribute 'OPC.UA.DA' := '0'}
	nCommand_Valve:	E_CRYO_BIN_ACT_CMD	:= E_CRYO_BIN_ACT_CMD.NONE;	// Command

	{attribute 'OPC.UA.DA' := '0'}
	bReset:		BOOL := FALSE;		// RESET Command

	{attribute 'OPC.UA.DA' := '0'}
	bValveCmd:	BOOL := FALSE;		// Valve Command - TRUE=OPEN, FALSE=CLOSE


	{attribute 'OPC.UA.DA' := '0'}
	timerTurbo:	TON;		// Timer for Turbo Pump
	
	{attribute 'OPC.UA.DA' := '0'}
	timerValveDelay:	TON;		// Timer for measuring time after Valve is closed
	
	{attribute 'OPC.UA.DA' := '0'}
	timerValveCtrl:	TON;		// Timer for Valve open/close timeout
	
	{attribute 'OPC.UA.DA' := '0'}
	trigEnable:	R_TRIG;			// Trigger for in_bEnable
	
	{attribute 'OPC.UA.DA' := '0'}
	trigDisable:F_TRIG;			// Trigger for in_bEnable=FALSE, i.e. Disable
	
	{attribute 'OPC.UA.DA' := '0'}
	trigTurbo:	R_TRIG;		// Trigger for start of TurboPump
	
	{attribute 'OPC.UA.DA' := '0'}
	trigValveClosed:	R_TRIG;		// Trigger for Valve Closed. Start timerValve on trigger.
	
END_VAR

// Increment cycle counter
stat.nCycleCounter := stat.nCycleCounter + 1;

// Pump control based on Valve status.
M_PumpCtrl();

// Check for errors
M_CheckErrors();

// Get Valve Command based on pressure and temperature conditions
M_SetValveCommand();


// Execute Valve FB on every cycle
Valve(	in_bExecute	:= bExecute_Valve,
		in_nCommand	:= nCommand_Valve,
		in_nFeedback:= in_nFeedback);


M_StateMachine();

METHOD M_CheckErrors
VAR_INPUT
END_VAR
VAR
END_VAR
// TODO: Set stat.sStatus for each failure
IF Valve.stat.bON  AND  (in_bRepressValveOpen  OR  NOT in_bRepressValveOK) THEN
	// Emergency situation. Close the Valve
	stat.bEmergency	:= TRUE;
	stat.bError	:= TRUE;
ELSIF stat.bEnabled  AND  (in_bRepressValveOpen  OR  NOT in_bRepressValveOK) THEN
	// The Evacuation system should never be enabled 
	// if there is a problem with the repressurizing valve.
	// Emergency situation. Do not operate.
	stat.bEmergency	:= TRUE;
	stat.bError	:= TRUE;
ELSIF NOT in_bRepressValveOK THEN
	stat.bError	:= TRUE;
ELSIF NOT in_Pressure_Cryo.bValid THEN
	stat.bError	:= TRUE;
ELSIF NOT in_Pressure_Evac.bValid THEN
	stat.bError	:= TRUE;
ELSIF Valve.stat.bError THEN
	stat.bError	:= TRUE;
ELSE
	stat.bError	:= FALSE;
END_IF

// Additional check for emergency situation.
// If there is an error while the Evacuation Valve is open, close it immediately.
IF stat.bError  AND  Valve.stat.bON  THEN
	stat.bEmergency	:= TRUE;
END_IF

IF stat.bError  THEN
	stat.bEnabled	:= FALSE;	// Disable Evacuation System
END_IF
END_METHOD

// Pump control based on Valve status.
METHOD M_PumpCtrl
VAR_INPUT
END_VAR
//
// Capture in_bEnable going TRUE.
// When it happens, start the pumps by activating the control output.
//
trigEnable(CLK:=in_bEnable);
IF trigEnable.Q THEN
	stat.bEnabled	:= TRUE;
	stat.bEmergency	:= FALSE;	// Clear emergency warning, if any
	stat.bError		:= FALSE;	// Clear error
	q_bPumpCtrl		:= TRUE;	// Start pumps
ELSIF NOT in_bEnable THEN
	stat.bEnabled		:= FALSE;
END_IF


//
// Set the status of the Root Pump
//
stat.bRootPumpON	:= i_bRootPumpOn;


//
// Set the status of the Turbo Pump
//
IF i_bTurboPumpOn THEN
	// Turbo pump is running.
	stat.bTurboPumpON	:= TRUE;
ELSE
	timerTurbo(IN:=FALSE);
	stat.bTurboPumpON		:= FALSE;
	stat.bTurboPump10min	:= FALSE;
END_IF



//
// Capture the moment when Turbo Pump started.
// Turbo Pump is fully operational after 10 min of operation (in_nTime_TurboPump).
//
// Execute timer for Turbo Pump
timerTurbo();

trigTurbo(CLK:=stat.bTurboPumpON);
IF trigTurbo.Q  THEN
	//
	// Turbo Pump has just started.
	// Start the timer that will signal that the turbo pump is fully operational.
	//
	// Reset the timer.
	timerTurbo(IN:=FALSE);
	// Start the timer for Turbo Pump warmup.
	timerTurbo(IN:=TRUE,PT:=UDINT_TO_TIME(in_Cryo_Cfg.nTime_TurboPump));
END_IF

IF timerTurbo.Q THEN
	// Turbo Pump is now fully operational.
	stat.bTurboPump10min	:= TRUE;
END_IF


//
// Capture the moment when the Valve is closed or the system is disabled.
// Pumps should be stopped in_nTime_DeltaTValve [ms] (e.g. 2000ms) after this event.
//
// Execute timer for Valve timer
timerValveDelay();


//
// Capture the moment when the valve is closed.
// Start the delay timer for in_Cryo_Cfg.nTime_DeltaTValve ms.
// After the delay, it is safe to stop the pumps.
//
trigValveClosed(CLK:=NOT stat.bValveOpen);
trigDisable(CLK:=stat.bEnabled);	// Falling edge of bEnable
IF trigValveClosed.Q OR trigDisable.Q  THEN
	// Reset the timer
	timerValveDelay(IN:=FALSE);
	// Start the Valve timer.
	timerValveDelay(IN:=TRUE,PT:=UDINT_TO_TIME(in_Cryo_Cfg.nTime_DeltaTValve));
END_IF


//
// The delay timer has expired.
// It is safe to stop the pumps.
//
IF timerValveDelay.Q THEN
	// Reset the timer
	timerValveDelay(IN:=FALSE);
	// Stop the pumps if evacuation is disabled
	IF NOT stat.bEnabled THEN
		q_bPumpCtrl	:= FALSE;
	END_IF
END_IF

// Update output var
stat.bValveOpen	:= Valve.stat.bON;
END_METHOD

METHOD M_SetStatus
VAR_INPUT
	nState:	E_CRYO_EVAC_SYS_STATE;
END_VAR
// TODO: Complete this


CASE nState OF
	
	E_CRYO_EVAC_SYS_STATE.OFF:
	stat.bDone	:= TRUE;
	stat.bBusy	:= FALSE;
	IF NOT stat.bError THEN
		stat.sState	:= 'OFF';
	END_IF
	stat.bActive	:= FALSE;
	
	E_CRYO_EVAC_SYS_STATE.ACTIVE_CLOSED:
	stat.bDone	:= TRUE;
	stat.bBusy	:= FALSE;
	IF NOT stat.bError THEN
		stat.sState	:= 'ACTIVE_OFF';
	END_IF
	stat.bActive	:= TRUE;
	
	E_CRYO_EVAC_SYS_STATE.ACTIVE_OPEN:
	stat.bDone	:= TRUE;
	stat.bBusy	:= FALSE;
	stat.bError	:= FALSE;
	stat.bActive	:= TRUE;
	stat.sState	:= 'ACTIVE_ON';
	
	E_CRYO_EVAC_SYS_STATE.ACTIVE_OPENING:
	stat.bDone	:= FALSE;
	stat.bBusy	:= TRUE;
	stat.bError	:= FALSE;
	stat.bActive	:= TRUE;
	stat.sState	:= 'ACTIVE_SWITCHING_ON...';
	
	E_CRYO_EVAC_SYS_STATE.ACTIVE_CLOSING:
	stat.bDone	:= FALSE;
	stat.bBusy	:= TRUE;
	stat.bError	:= FALSE;
	stat.bActive	:= TRUE;
	stat.sState	:= 'ACTIVE_SWITCHING_OFF...';
	
	E_CRYO_EVAC_SYS_STATE.ERROR:
	stat.bDone	:= TRUE;
	stat.bBusy	:= FALSE;
//	stat.bError	:= TRUE;
	stat.bActive	:= FALSE;
//	stat.sState	:= 'ERROR';

END_CASE
END_METHOD

//
// Determines if the valve should be open or closed.
// It sets the internal variable nCommand_Valve.
//
METHOD M_SetValveCommand
VAR_INPUT
END_VAR
// Reset bExecute_Valve flag and the Valve command.
// They might be set again depending on the bEnable flag and the environmental conditions.
bExecute_Valve	:= FALSE;
nCommand_Valve	:= E_CRYO_BIN_ACT_CMD.NONE;


// 
// Set the Valve command based on temperature and pressure.
// If the system is not enabled or there is an error, the valve should be closed.
//
IF stat.bError THEN
	// Close the Valve on any error.
	nCommand_Valve	:= E_CRYO_BIN_ACT_CMD.OFF;
ELSIF NOT stat.bEnabled THEN
	// Close the Valve if the system is Disabled/OFF.
	nCommand_Valve	:= E_CRYO_BIN_ACT_CMD.OFF;
ELSIF 	(in_Pressure_Cryo.lrPressure > in_Cryo_Cfg.lrPress_Atm)  AND  
		(in_Temp_Cryo.lrTempK > in_Cryo_Cfg.lrTemp_Warm) THEN
	// Cryo is Warm and Pressurized - safe to open Valve.
	nCommand_Valve	:= E_CRYO_BIN_ACT_CMD.ON;
//ELSIF NOT in_Pressure_Cryo.bInVacuum THEN
ELSIF in_Pressure_Cryo.lrPressure >= in_Cryo_Cfg.lrPress_InVac THEN
	// If not in vacuum, it means the cryostat must be WARM.
	IF (in_Pressure_Evac.lrPressure < in_Pressure_Cryo.lrPressure) THEN
		nCommand_Valve	:= E_CRYO_BIN_ACT_CMD.ON;
	END_IF
ELSIF in_Temp_Cryo.lrTempK < in_Cryo_Cfg.lrTemp_Precooled THEN
	// Cryostat is COLD.
	IF ((in_Pressure_Evac.lrPressure < in_Pressure_Cryo.lrPressure) AND stat.bTurboPumpON) OR  
		(stat.bTurboPump10min AND in_Pressure_Evac.lrPressure < 7.0E-5) THEN
		nCommand_Valve	:= E_CRYO_BIN_ACT_CMD.ON;
	END_IF
//ELSIF in_Pressure_Cryo.bInVacuum THEN
ELSIF in_Pressure_Cryo.lrPressure < in_Cryo_Cfg.lrPress_InVac THEN
	// Cryostat is in vacuum.
	IF (in_Pressure_Evac.lrPressure < in_Pressure_Cryo.lrPressure)  AND stat.bTurboPumpON THEN
		nCommand_Valve	:= E_CRYO_BIN_ACT_CMD.ON;
	END_IF
END_IF


//
// Apply Valve command depending on the Evacuation System state.
// Update the State as well.
//
IF (stat.bError OR stat.bEmergency) AND stat.nState	<> E_CRYO_EVAC_SYS_STATE.ACTIVE_CLOSING THEN
	//
	// There is an error or emergency in the system. 
	// Close the valve. 
	//
	// Trigger Valve closing
	bExecute_Valve	:= TRUE;
	nCommand_Valve	:= E_CRYO_BIN_ACT_CMD.OFF;
	Valve(in_bExecute	:= FALSE);
	Valve(in_bExecute	:= TRUE, in_nCommand := nCommand_Valve);
	stat.nState	:= E_CRYO_EVAC_SYS_STATE.ACTIVE_CLOSING;
ELSIF stat.nState = E_CRYO_EVAC_SYS_STATE.ACTIVE_CLOSED  THEN 
	IF  nCommand_Valve = E_CRYO_BIN_ACT_CMD.ON THEN
		bExecute_Valve	:= TRUE;
		timerValveCtrl(IN:=FALSE);
		timerValveCtrl(IN:=TRUE, PT:=UDINT_TO_TIME(in_nTimeout));
		stat.nState	:= E_CRYO_EVAC_SYS_STATE.ACTIVE_OPENING;
	ELSE
		bExecute_Valve	:= FALSE;
		IF stat.bEnabled THEN
			stat.nState	:= E_CRYO_EVAC_SYS_STATE.ACTIVE_CLOSED;
		ELSE
			stat.nState	:= E_CRYO_EVAC_SYS_STATE.OFF;
		END_IF
	END_IF
ELSIF stat.nState	= E_CRYO_EVAC_SYS_STATE.ACTIVE_OPEN  THEN 
	IF  nCommand_Valve = E_CRYO_BIN_ACT_CMD.OFF  OR  NOT stat.bEnabled  THEN
		bExecute_Valve	:= TRUE;
		timerValveCtrl(IN:=FALSE);
		timerValveCtrl(IN:=TRUE, PT:=UDINT_TO_TIME(in_nTimeout));
		stat.nState	:= E_CRYO_EVAC_SYS_STATE.ACTIVE_CLOSING;
	ELSE
		bExecute_Valve	:= FALSE;
		stat.nState	:= E_CRYO_EVAC_SYS_STATE.ACTIVE_OPEN;
	END_IF
END_IF
END_METHOD

METHOD M_StateMachine
VAR_INPUT
END_VAR
CASE stat.nState OF
	/////////////////////////////////
	E_CRYO_EVAC_SYS_STATE.NONE:
	/////////////////////////////////
	//
	// This is the state on power-up.
	// Determine the initial state based on the command and actuator state.
	IF NOT stat.bEnabled THEN
		IF Valve.stat.bOFF  AND  NOT stat.bRootPumpON AND NOT stat.bTurboPumpON THEN
			stat.nState	:= E_CRYO_EVAC_SYS_STATE.OFF;
		END_IF
	ELSE
		IF	stat.bError	THEN
			IF Valve.stat.bON THEN
				stat.nState	:= E_CRYO_EVAC_SYS_STATE.EMERGENCY;
			ELSE
				stat.nState	:= E_CRYO_EVAC_SYS_STATE.ERROR;
			END_IF
			stat.nState	:= E_CRYO_EVAC_SYS_STATE.ERROR;
		ELSIF Valve.stat.bON THEN
			stat.nState	:= E_CRYO_EVAC_SYS_STATE.ACTIVE_OPEN;
		ELSIF Valve.stat.bOFF  THEN
			stat.nState	:= E_CRYO_EVAC_SYS_STATE.ACTIVE_CLOSED;
		END_IF
	END_IF
	M_SetStatus(stat.nState);	
	RETURN;
	

	/////////////////////////////////
	E_CRYO_EVAC_SYS_STATE.OFF:
	/////////////////////////////////
	//
	IF stat.bEnabled  THEN
		// Set next state.
		stat.nState	:= E_CRYO_EVAC_SYS_STATE.ACTIVE_CLOSED;
	END_IF
	M_SetStatus(stat.nState);	
	RETURN;
	
	
	////////////////////////////////////////
	E_CRYO_EVAC_SYS_STATE.ACTIVE_CLOSING:
	////////////////////////////////////////
	//
	timerValveCtrl();
	IF timerValveCtrl.Q THEN
		// Closing failure
		stat.bCtrlOK	:= FALSE;
		stat.sStatus	:= 'Valve failed to close';
		stat.bError	:= TRUE;
		stat.nState	:= E_CRYO_EVAC_SYS_STATE.ERROR;
	ELSIF NOT stat.bValveOpen THEN
		timerValveCtrl(IN:=FALSE);
		// Set next state.
		stat.nState	:= E_CRYO_EVAC_SYS_STATE.ACTIVE_CLOSED;
	END_IF
	M_SetStatus(stat.nState);	
	RETURN;
	
	
	////////////////////////////////////////
	E_CRYO_EVAC_SYS_STATE.ACTIVE_CLOSED:
	////////////////////////////////////////
	//
	IF	NOT stat.bEnabled  THEN
		// Set next state
		stat.nState	:= E_CRYO_EVAC_SYS_STATE.OFF;
	ELSIF stat.bValveOpen THEN
		// Set next state.
		stat.nState	:= E_CRYO_EVAC_SYS_STATE.ACTIVE_OPEN;
	END_IF
	M_SetStatus(stat.nState);	
	RETURN;
	
	
	////////////////////////////////////////
	E_CRYO_EVAC_SYS_STATE.ACTIVE_OPENING:
	////////////////////////////////////////
	//
	timerValveCtrl();
	IF timerValveCtrl.Q THEN
		// Closing failure
		stat.bCtrlOK	:= FALSE;
		stat.sStatus	:= 'Valve failed to open';
		stat.bError	:= TRUE;
		stat.nState	:= E_CRYO_EVAC_SYS_STATE.ERROR;
	ELSIF stat.bValveOpen THEN
		timerValveCtrl(IN:=FALSE);
		// Set next state.
		stat.nState	:= E_CRYO_EVAC_SYS_STATE.ACTIVE_OPEN;
	END_IF
	M_SetStatus(stat.nState);	
	RETURN;
	
	
	//////////////////////////////////////////
	E_CRYO_EVAC_SYS_STATE.ACTIVE_OPEN:
	//////////////////////////////////////////
	//
	IF NOT stat.bValveOpen THEN
		// Set next state.
		stat.nState	:= E_CRYO_EVAC_SYS_STATE.ACTIVE_CLOSED;
	END_IF
	M_SetStatus(stat.nState);	
	RETURN;
	

	///////////////////////////////////////////
	E_CRYO_EVAC_SYS_STATE.EMERGENCY:
	///////////////////////////////////////////
	//
	IF Valve.stat.bOFF THEN
		// The actuator is OFF, transition completed.
		// Goto Active_Off.
		stat.nState	:= E_CRYO_EVAC_SYS_STATE.ACTIVE_CLOSED;
	END_IF
	M_SetStatus(stat.nState);	
	RETURN;
	
	/////////////////////////////////
	E_CRYO_EVAC_SYS_STATE.ERROR:
	/////////////////////////////////
	//
	M_User_TryRecovery();

END_CASE
END_METHOD

METHOD M_TrgValveClosure : BOOL
VAR_INPUT
END_VAR
END_METHOD

METHOD M_User_TryRecovery
VAR_INPUT
END_VAR
// TODO USER
// This is the default recovery routine.
// To be customided by the user, if needed.
//
IF bReset THEN
	// RESET the controller in order to try to clear error
	bReset	:= FALSE;	// Clear RESET flag
	
	// Trigger action
	Valve(in_bExecute:=FALSE);
	Valve(in_bExecute:=TRUE, in_nCommand:=E_CRYO_BIN_ACT_CMD.OFF);
	
	// Goto SWITCHING_OFF state
	stat.nState	:= E_CRYO_EVAC_SYS_STATE.ACTIVE_CLOSING;
	M_SetStatus(stat.nState);	
ELSIF NOT Valve.stat.bError AND stat.bCtrlOK  THEN
	// Self recovery since everything seems to be OK now.
	// Goto NONE state.
	// From there proper state will be found and set.
	stat.nState	:= E_CRYO_EVAC_SYS_STATE.NONE;
	M_SetStatus(stat.nState);	
END_IF
END_METHOD

END_FUNCTION_BLOCK

// POUs/Simulation/FB_CRYO_SIM_TEMPERATURE
//
// This FB simulates temperature in degK.
//
FUNCTION_BLOCK FB_CRYO_SIM_TEMPERATURE
VAR_INPUT
	in_lrScale:		LREAL 	:= 0.1;		// Scale factor, T = raw * scale. Default 0.1
	in_lrTempK:		LREAL	:= 283.15;	// Start Temperature [K]
	in_lrTempDelta:	LREAL	:= 11.25;	// Delta Temperature +- for SINE wave [K]
	in_nPeriod:		UDINT	:= 10000;	// RAMP/SINE Command period, default 10000ms = 10s
	in_bAutoSine:	BOOL	:= FALSE;	// Flag if SINE wave should start immediately
	
END_VAR
VAR
	q_nStatus	AT%Q*:	UINT	:= 0;	// Simulated status
	q_nValue	AT%Q*:	INT		:= 100;	// Simulated value [bit]
	
	{attribute 'OPC.UA.DA' := '0'}
	bStarted:		BOOL := FALSE;
	{attribute 'OPC.UA.DA' := '0'}
	toggleTimer:	TON;		// Timer for PDO (alive) toggle
	{attribute 'OPC.UA.DA' := '0'}
	rampTimer:		TON;		// Timer for temperature ramp

	{attribute 'OPC.UA.DA' := '0'}
	nToggleMask:	UINT := 2#1000_0000_0000_0000;

	lrTempK:		LREAL	:= 283.15;	// Simulated temperature [K]
	{attribute 'OPC.UA.DA' := '0'}
	lrTempStart:	LREAL	:= 283.15;	// Simulated temperature start [K]
	{attribute 'OPC.UA.DA' := '0'}
	lrTempEnd:		LREAL	:= 0.0;		// Simulated temperature end   [K]
	{attribute 'OPC.UA.DA' := '0'}
	lrTempDelta:	LREAL	:= 11.25;	// Delta Temperature +- for SINE wave [K]
	{attribute 'OPC.UA.DA' := '0'}
	nValue:			INT		:= 100;		// Simulated value [bit]

	{attribute 'OPC.UA.DA' := '0'}
	nPeriod:		UDINT	:= 10000;	// RAMP/SINE Command period, default 10000ms = 10s
	
	{attribute 'OPC.UA.DA' := '0'}
	nState:		INT	:= SIM_TEMP_STATE_FIXED;
	
END_VAR
VAR CONSTANT 
	{attribute 'OPC.UA.DA' := '0'}
    SIM_TEMP_STATE_NONE:	INT :=  0;
	{attribute 'OPC.UA.DA' := '0'}
    SIM_TEMP_STATE_FIXED:	INT := 10;
	{attribute 'OPC.UA.DA' := '0'}
    SIM_TEMP_STATE_RAMP:	INT := 20;
	{attribute 'OPC.UA.DA' := '0'}
    SIM_TEMP_STATE_SINE:	INT := 30;
	
	{attribute 'OPC.UA.DA' := '0'}
    SIM_TEMP_RAMP_UP:		INT := 0;
	{attribute 'OPC.UA.DA' := '0'}
    SIM_TEMP_RAMP_DOWN:		INT := 1;
	
END_VAR

//
// Simulate terminal alive toggle every 160ms.
//
IF NOT bStarted THEN
	bStarted	:= TRUE;
	lrTempK		:= in_lrTempK;	// Assign starting value
	lrTempDelta	:= in_lrTempDelta;
	nPeriod		:= in_nPeriod;
	IF in_bAutoSine THEN
		M_StartSine(in_lrValueStart:=lrTempK,
					in_lrValueDelta:=lrTempDelta,
					in_nPeriod:=nPeriod);
	END_IF
	toggleTimer(IN:=FALSE);
END_IF
toggleTimer(IN:=TRUE,PT:=T#160MS);

IF toggleTimer.Q THEN
	q_nStatus	:= q_nStatus XOR nToggleMask;
	// Restart the timer
	toggleTimer(IN:=FALSE);
END_IF


//
// Handle states 
//
IF nState = SIM_TEMP_STATE_RAMP THEN
	rampTimer(IN:=TRUE);
	lrTempK	:=	lrTempStart + 
				(lrTempEnd - lrTempStart)* TIME_TO_LREAL(rampTimer.ET)/TIME_TO_LREAL(rampTimer.PT);
	IF rampTimer.Q THEN
		rampTimer(IN:=FALSE);
		nState	:= SIM_TEMP_STATE_FIXED;
	END_IF
ELSIF nState = SIM_TEMP_STATE_SINE THEN
	rampTimer(IN:=TRUE);
	lrTempK	:=	lrTempStart + 
				lrTempDelta * SIN(2 * PI * TIME_TO_LREAL(rampTimer.ET)/TIME_TO_LREAL(rampTimer.PT));
	IF rampTimer.Q THEN
		rampTimer(IN:=FALSE);
		// Continue with the sine wave.
		rampTimer(IN:=TRUE,PT:=UDINT_TO_TIME(nPeriod));
	END_IF
END_IF



//
// Set the raw reading, i.e. K -> bit.
//
q_nValue	:= M_degK2bit(lrTempK);

METHOD M_bit2degK : LREAL
VAR_INPUT
	in_nValue:	INT;
END_VAR
//
// Set the raw reading, i.e. K -> bit.
// Conversion is K -> C -> bit.
//
M_bit2degK	:= in_nValue * in_lrScale + 273.15;
END_METHOD

METHOD M_degK2bit : INT
VAR_INPUT
	in_lrValue:	LREAL;
END_VAR
//
// Set the raw reading, i.e. K -> bit.
// Conversion is K -> C -> bit.
//
M_degK2bit	:= LREAL_TO_INT((in_lrValue - 273.15) / in_lrScale);
END_METHOD

METHOD M_RampTo
VAR_INPUT
	in_lrValueEnd:		LREAL;
	in_nPeriod:			UDINT	:= 10000;	// RAMP/SINE Command period, default 10000ms = 10s
END_VAR
rampTimer(IN:=FALSE);
rampTimer(IN:=TRUE,PT:=UDINT_TO_TIME(in_nPeriod));
lrTempStart	:= lrTempK;
lrTempEnd	:= in_lrValueEnd;
nPeriod		:= in_nPeriod;
nState		:= SIM_TEMP_STATE_RAMP;
END_METHOD

METHOD M_SetValue
VAR_INPUT
	in_lrValue:	LREAL;
END_VAR
rampTimer(IN:=FALSE);
lrTempK	:= in_lrValue;
nState	:= SIM_TEMP_STATE_FIXED;
END_METHOD

METHOD M_StartRamp
VAR_INPUT
	in_lrValueStart:	LREAL;
	in_lrValueEnd:		LREAL;
	in_nPeriod:			UDINT	:= 10000;	// RAMP/SINE Command period, default 10000ms = 10s
END_VAR
rampTimer(IN:=FALSE);
rampTimer(IN:=TRUE,PT:=UDINT_TO_TIME(in_nPeriod));
lrTempStart	:= in_lrValueStart;
lrTempEnd	:= in_lrValueEnd;
nPeriod		:= in_nPeriod;
nState		:= SIM_TEMP_STATE_RAMP;
END_METHOD

METHOD M_StartSine
VAR_INPUT
	in_lrValueStart:	LREAL;
	in_lrValueDelta:	LREAL;
	in_nPeriod:			UDINT	:= 10000;	// RAMP/SINE Command period, default 10000ms = 10s
END_VAR
rampTimer(IN:=FALSE);
rampTimer(IN:=TRUE,PT:=UDINT_TO_TIME(in_nPeriod));
lrTempStart	:= in_lrValueStart;
lrTempDelta	:= in_lrValueDelta;
nPeriod		:= in_nPeriod;
nState		:= SIM_TEMP_STATE_SINE;
END_METHOD

METHOD M_Stop
VAR_INPUT
END_VAR
// Stop ramping.
// Keep value as it is.
rampTimer(IN:=FALSE);
nState	:= SIM_TEMP_STATE_FIXED;
END_METHOD

END_FUNCTION_BLOCK

// POUs/Simulation/FB_CRYO_SIM_PRESSURE
//
// This FB simulates pressure.
//
FUNCTION_BLOCK FB_CRYO_SIM_PRESSURE
VAR_INPUT
	in_nType:	E_CRYO_SENSOR_TYPE_PRESS;
	// Scale factor bits -> Volt, U = raw / scale. 
	// Default for 16-bit, +-10V or 0..10V AI: 2^16/10/2 = 3276.8 bit
	in_lrBitsPerVolt:	LREAL := 3276.8;	// Scale factor, U = raw / scale. Default 3276.8
	in_lrPress:		LREAL	:= 777.0;	// Starting Pressure
	in_nPeriod:		UDINT	:= 10000;	// RAMP Command period, default 10000ms = 10s
	
END_VAR
VAR
	q_nStatus	AT%Q*:	UINT	:= 0;		// Simulated status
	q_nValue	AT%Q*:	INT		:= 27953;	// Simulated value [bit] = 777 mbar
	
	{attribute 'OPC.UA.DA' := '0'}
	bStarted:		BOOL := FALSE;
	{attribute 'OPC.UA.DA' := '0'}
	toggleTimer:	TON;		// Timer for PDO (alive) toggle
	{attribute 'OPC.UA.DA' := '0'}
	rampTimer:		TON;		// Timer for temperature ramp

	{attribute 'OPC.UA.DA' := '0'}
	nToggleMask:	UINT := 2#1000_0000_0000_0000;

	lrPress:		LREAL	:= 777.0;	// Simulated Pressure
	{attribute 'OPC.UA.DA' := '0'}
	lrPressStart:	LREAL	:= 0.0;		// Simulated Pressure start[mbar]
	{attribute 'OPC.UA.DA' := '0'}
	lrPressEnd:		LREAL	:= 0.0;		// Simulated Pressure end  [mbar]
	{attribute 'OPC.UA.DA' := '0'}
	lrPressDelta:	LREAL	:= 0.0;		// Simulated Pressure delta for curve  [mbar]
	{attribute 'OPC.UA.DA' := '0'}
	lrCurveScale:	LREAL	:= 0.3;		// t^lrCurveScale factor
	{attribute 'OPC.UA.DA' := '0'}
	nValue:			INT		:= 27953;	// Simulated value [bit]
	{attribute 'OPC.UA.DA' := '0'}
	nPeriod:		UDINT	:= 10000;	// RAMP Command period, default 10000ms = 10s
	
	{attribute 'OPC.UA.DA' := '0'}
	State:		INT	:= SIM_VACUUM_STATE_FIXED;
	
	// Temporary variables
	{attribute 'OPC.UA.DA' := '0'}
	lrTmp1:		LREAL;
	
END_VAR
VAR CONSTANT 
	{attribute 'OPC.UA.DA' := '0'}
    SIM_VACUUM_STATE_NONE:	INT :=  0;
	{attribute 'OPC.UA.DA' := '0'}
    SIM_VACUUM_STATE_FIXED:	INT := 10;
	{attribute 'OPC.UA.DA' := '0'}
    SIM_VACUUM_STATE_RAMP:	INT := 20;
	{attribute 'OPC.UA.DA' := '0'}
    SIM_VACUUM_STATE_CURVE:	INT := 30;
	
	{attribute 'OPC.UA.DA' := '0'}
    SIM_VACUUM_RAMP_UP:		INT := 0;
	{attribute 'OPC.UA.DA' := '0'}
    SIM_VACUUM_RAMP_DOWN:	INT := 1;
	
END_VAR

//
// Simulate terminal alive toggle every 160ms.
//
IF NOT bStarted THEN
	bStarted	:= TRUE;
	lrPress		:= in_lrPress;
	nPeriod		:= in_nPeriod;
	toggleTimer(IN:=FALSE);
END_IF
toggleTimer(IN:=TRUE,PT:=T#160MS);

IF toggleTimer.Q THEN
	q_nStatus	:= q_nStatus XOR nToggleMask;
	// Restart the timer
	toggleTimer(IN:=FALSE);
END_IF



//
// Handle states
//
rampTimer(IN:=TRUE);
IF State = SIM_VACUUM_STATE_RAMP THEN
	lrPress	:=	lrPressStart + 
				(lrPressEnd - lrPressStart)* TIME_TO_LREAL(rampTimer.ET)/TIME_TO_LREAL(rampTimer.PT);
	IF rampTimer.Q THEN
		rampTimer(IN:=FALSE);
		State	:= SIM_VACUUM_STATE_FIXED;
	END_IF
ELSIF State = SIM_VACUUM_STATE_CURVE THEN
	lrTmp1	:= TIME_TO_LREAL(rampTimer.ET)/TIME_TO_LREAL(rampTimer.PT);
	lrTmp1	:= EXPT(lrTmp1,lrCurveScale);
	lrPress	:=	lrPressStart + (lrPressEnd - lrPressStart)* lrTmp1;
	IF rampTimer.Q THEN
		rampTimer(IN:=FALSE);
		State	:= SIM_VACUUM_STATE_FIXED;
	END_IF
END_IF


//
// Set the raw reading, i.e. mbar -> bit.
// Conversion is mbar -> Volt -> bit.
//
IF lrPress > 0.0  THEN
	q_nValue	:= M_mbar2bit(lrPress);
END_IF

METHOD M_bit2mbar : LREAL
VAR_INPUT
	in_nBits:	INT;
END_VAR
VAR
	lrVoltage:	LREAL;
	lrPressure:	LREAL;
END_VAR
lrVoltage	:= in_nBits / in_lrBitsPerVolt;

CASE in_nType OF 
	E_CRYO_SENSOR_TYPE_PRESS.PKR_250,
	E_CRYO_SENSOR_TYPE_PRESS.PKR_360:
		// Conversion Volt -> mbar.
		// Pfeiffer PKR250/251
		// P = 10^(C1 * U - C2).
		// C1 = 1.667, C2 = d = 11.33
		// P = 10^(1.667 * U - 11.33)
		// U = (log(P)+C2)/C1
		// U = (log(P)+11.33)/1.667
		lrPressure	:= EXPT(10.0, (1.667 * lrVoltage - 11.33));
	E_CRYO_SENSOR_TYPE_PRESS.CMR_361:
		// Conversion Volt -> mbar.
		// Pfeiffer CMR361
		// P = (U - 1) * C1 * C2 [mbar]
		// C1 = 0.125, C2=FullScale = 1000 
		// P = (U - 1) * 0.125 * 1000.0 = (U-1) * 125[mbar]
		// P = (U-1) * 125
		// U = P/125 + 1
		lrPressure	:= (lrVoltage - 1) * 125;
	E_CRYO_SENSOR_TYPE_PRESS.WRG_D_NW25:
		// Edwards WRG-D-NW25 Conversion Volt -> mbar.
		// Range 10^-9 .. 100
		// P = 10^(C1 * U - C2).
		// P = 10^(1.5 * U - 12.0)
		// Valid range for U is 2.0-10.0
		lrPressure	:= EXPT(10.0, (1.5 * lrVoltage - 12.0));
END_CASE

M_bit2mbar	:= lrPressure;
END_METHOD

METHOD M_mbar2bit : INT
VAR_INPUT
	in_lrValue:	LREAL;
END_VAR
VAR
	lrValue:	LREAL;
	lrVoltage:	LREAL;
END_VAR
// Pressure cannot be zero
lrValue := MAX(1.0E-9,in_lrValue);

CASE in_nType OF 
	E_CRYO_SENSOR_TYPE_PRESS.PKR_250,
	E_CRYO_SENSOR_TYPE_PRESS.PKR_360:
		// Conversion Volt -> mbar.
		// Pfeiffer PKR250/251
		// P = 10^(C1 * U - C2).
		// C1 = 1.667, C2 = d = 11.33
		// P = 10^(1.667 * U - 11.33)
		// U = (log(P)+C2)/C1
		// U = (log(P)+11.33)/1.667
		lrVoltage	:= (LOG(lrValue) + 11.33) / 1.667;
	E_CRYO_SENSOR_TYPE_PRESS.CMR_361:
		// Conversion Volt -> mbar.
		// Pfeiffer CMR361
		// P = (U - 1) * C1 * C2 [mbar]
		// C1 = 0.125, C2=FullScale = 1000 
		// P = (U - 1) * 0.125 * 1000.0 = (U-1) * 125[mbar]
		// P = (U-1) * 125
		// U = P/125 + 1
		lrVoltage	:= lrValue/125 + 1.0;
	E_CRYO_SENSOR_TYPE_PRESS.WRG_D_NW25:
		// Edwards WRG-D-NW25 Conversion Volt -> mbar.
		// Range 10^-9 .. 100
		// P = 10^(C1 * U - C2).
		// P = 10^(1.5 * U - 12.0)
		// Valid range for U is 2.0-10.0
		lrVoltage	:= (LOG(lrValue) + 12.0) / 1.5;
END_CASE

M_mbar2bit	:= LREAL_TO_INT(lrVoltage * in_lrBitsPerVolt);
END_METHOD

METHOD M_RampTo
VAR_INPUT
	in_lrValueEnd:		LREAL;
	in_nPeriod:			UDINT	:= 10000;	// RAMP/SINE Command period, default 10000ms = 10s
END_VAR
rampTimer(IN:=FALSE);
rampTimer(IN:=TRUE,PT:=UDINT_TO_TIME(in_nPeriod));
lrPressStart	:= lrPress;
lrPressEnd		:= in_lrValueEnd;
nPeriod			:= in_nPeriod;
State			:= SIM_VACUUM_STATE_RAMP;
END_METHOD

METHOD M_SetValue
VAR_INPUT
	in_lrValue:	LREAL;
END_VAR
rampTimer(IN:=FALSE);
lrPress	:= in_lrValue;
State	:= SIM_VACUUM_STATE_FIXED;
END_METHOD

METHOD M_StartCurve
VAR_INPUT
	in_lrValueEnd:		LREAL;
	in_nPeriod:			UDINT	:= 20000;	// RAMP/SINE Command period, default 10000ms = 10s
	in_lrCurveScale:	LREAL	:= 0.3;		// t^lrCurveScale factor
END_VAR
rampTimer(IN:=FALSE);
rampTimer(IN:=TRUE,PT:=UDINT_TO_TIME(in_nPeriod));
lrPressStart	:= lrPress;
lrPressEnd		:= in_lrValueEnd;
lrCurveScale	:= in_lrCurveScale;
State			:= SIM_VACUUM_STATE_CURVE;
END_METHOD

METHOD M_StartRamp
VAR_INPUT
	in_lrValueStart:	LREAL;
	in_lrValueEnd:		LREAL;
END_VAR
rampTimer(IN:=FALSE);
rampTimer(IN:=TRUE,PT:=UDINT_TO_TIME(nPeriod));
lrPressStart	:= in_lrValueStart;
lrPressEnd		:= in_lrValueEnd;
State			:= SIM_VACUUM_STATE_RAMP;
END_METHOD

METHOD M_Stop
VAR_INPUT
END_VAR
// Stop ramping.
// Keep value as it is.
rampTimer(IN:=FALSE);
State	:= SIM_VACUUM_STATE_FIXED;
END_METHOD

END_FUNCTION_BLOCK

// POUs/Simulation/FB_CRYO_SIM_SBG232
FUNCTION_BLOCK FB_CRYO_SIM_SBG232
VAR_INPUT
	in_lrRefTemp:	LREAL := 21.0;	// Temperature reference point [°C]
	in_lrRefFlow:	LREAL := 4.30;	// Flow reference point [L/min]
	in_lrVarTemp:	LREAL := 2.0;	// Temperature reading variation [°C]
	in_lrVarFlow:	LREAL := 0.1;	// Flow reading variation [L/min]
END_VAR
VAR_OUTPUT
END_VAR
VAR
	temp:	FB_CRYO_SIM_SINE;	// Temperature variation as sine wave
	flow:	FB_CRYO_SIM_SINE;	// Flow variation as sine wave
	
	lrTemp:	LREAL;
	lrFlow:	LREAL;
	nWord:	WORD;
	
	q_nCouplerState			AT %Q*:	UINT	:= 8;
	q_nDeviceStateInputCh	AT %Q*:	USINT	:= 3;
	q_ArrPortProcessData	AT %Q*:	ARRAY [0..3] OF BYTE;
END_VAR

// Simulate temperature and flow variations as sinewaves
temp(in_lrAmplitude:=in_lrVarTemp, in_nPeriod:=60000);
flow(in_lrAmplitude:=in_lrVarFlow, in_nPeriod:=120000);

// Calculate simulated values
lrTemp	:= in_lrRefTemp + temp.out_lrValue;
lrFlow	:= in_lrRefFlow + flow.out_lrValue;


// Set output variables

////////////////
// Temperature
////////////////

// lrVal	:= TRUNC(256.0 * i_ArrPortProcessData[2] + i_ArrPortProcessData[3]) / 4;	// /4 = SHR(2)
nWord	:= LREAL_TO_WORD(lrTemp	* 4);
q_ArrPortProcessData[2]	:= UINT_TO_BYTE(16#FF AND SHR(nWord,8));
q_ArrPortProcessData[3]	:= UINT_TO_BYTE(16#FF AND nWord);


//////////////
// Flow
//////////////

// lrVal	:= (256.0 * i_ArrPortProcessData[0] + i_ArrPortProcessData[1]) / 100.0;
nWord	:= LREAL_TO_WORD(lrFlow	* 100.0);
q_ArrPortProcessData[0]	:= UINT_TO_BYTE(16#FF AND SHR(nWord,8));
q_ArrPortProcessData[1]	:= UINT_TO_BYTE(16#FF AND nWord);

END_FUNCTION_BLOCK

// POUs/Simulation/FB_CRYO_SIM_SINE
// Simulator that generates sine wave 
FUNCTION_BLOCK FB_CRYO_SIM_SINE
VAR_INPUT
	in_lrAmplitude:	LREAL := 1.0;
	in_nPeriod:		UDINT := 10000;
END_VAR
VAR_OUTPUT
	out_lrValue:	LREAL;
END_VAR
VAR
	
	{attribute 'OPC.UA.DA':='0'}
	timer:			TON;
	
	{attribute 'OPC.UA.DA':='0'}
	bInitialised:	BOOL := FALSE;		// Used to start timer for the first time
	
	{attribute 'OPC.UA.DA':='0'}
	i:	INT;

END_VAR
VAR_TEMP
	t1:	LREAL;
	t2:	LREAL;
	t3:	LREAL;
	t4:	LREAL;
END_VAR

// Check possible devision by zero
IF in_nPeriod = 0 THEN
	in_nPeriod	:= 1000;
END_IF

IF NOT bInitialised THEN
	bInitialised := TRUE;
	
	// Start timer for signal=FALSE
	timer(IN:=FALSE);
	timer(IN:=TRUE, PT:=UDINT_TO_TIME(in_nPeriod));
	RETURN;
END_IF

// Execute timer
// The timer is actually used just for the 'angle' for the sin().
// Angle = ET / PT * 2PI
timer();

// If the timer expired, just restart it
IF timer.Q THEN
		timer(IN:=FALSE);
		timer(IN:=TRUE, PT:=UDINT_TO_TIME(in_nPeriod));
END_IF

// Set the output
t1	:= TIME_TO_LREAL(timer.ET);
t2	:= TIME_TO_LREAL(timer.PT);
t3	:= t1 / t2 * 2 * 3.14;
t4	:= in_lrAmplitude * SIN(t3);

// Set output
out_lrValue	:= t4;

END_FUNCTION_BLOCK

// POUs/Subsystems/Evacuation/FB_CRYO_EVAC_BASE
FUNCTION_BLOCK FB_CRYO_EVAC_BASE
VAR_INPUT
	in_bEnable:					BOOL := FALSE;	// System active while in_bEnable is TRUE
	in_lrCryoPressure:			LREAL;			// Cryo pressure
END_VAR
VAR_OUTPUT
END_VAR
VAR
	rpRef:	REFERENCE TO FB_CRYO_PUMP_BASE;		// Roughing Pump
	tpRef:	REFERENCE TO FB_CRYO_PUMP_BASE;		// Turbo Molecular Pump
	valve:	FB_CRYO_VALVE_CTRL;					// Insulation Valve
	
	press1:	FB_CRYO_SENSOR_PRESSURE;	// Prevacuum pressure gauge #1
	press2:	FB_CRYO_SENSOR_PRESSURE;	// Prevacuum pressure gauge #2
	prevac:	FB_CRYO_PRESSURE_VOTE;		// Prevacuum pressure 
	
	cfg:	T_CRYO_EVAC_CFG;
	ctrl:	T_CRYO_EVAC_CTRL;
	stat:	T_CRYO_EVAC_STAT;
	
	timer:	TON;
	trig:	R_TRIG;	// Start trigger
END_VAR

// NOTE: Configuration is set on the first cycle.
//       Once stat.bConfigured is TRUE, 
//       configuration is not updated any more.
M_Configure();

M_ReadSensors();

M_ExecuteControllers();

M_UpdateStatus();

M_StateMachine();

METHOD M_Activity_ClosingValve
VAR_INPUT
END_VAR
IF valve.stat.bActOFF THEN
	// The valve is closed.
	// Apply a delay before stopping Turbo pump.
	// Start the timer for the delay.
	timer(IN:=FALSE);
	timer(IN:=TRUE, PT:=cfg.tDelay);
	stat.nState	:= E_CRYO_EVAC_STATE.DELAY_STOPPING;	// Next state
	M_SetLabels();
END_IF
END_METHOD

METHOD M_Activity_DelayBeforeStoppingPumps
VAR_INPUT
END_VAR
timer();

IF timer.Q THEN
	// Delay timer expired.
	// Reset timer.
	timer(IN:=FALSE);
	
	// Stop Turbo Pump.
	ctrl.bEnable_TP	:= FALSE;
	stat.nState		:= E_CRYO_EVAC_STATE.STOP_T_PUMP;	// Next state
	M_SetLabels();
END_IF
END_METHOD

METHOD M_Activity_Evacuating
VAR_INPUT
END_VAR
// System is started by setting in_bEnable to TRUE
IF NOT in_bEnable THEN
	// If system is disabled, start stopping procedure.
	ctrl.bEnable_Valve	:= FALSE;
	stat.nState			:= E_CRYO_EVAC_STATE.CLOSE_INSULATION_VALVE;	// Next state
	M_SetLabels();
ELSIF prevac.stat.lrPressure > cfg.lrThld_Prevac THEN
	// Something is wrong. Prevacuum pressure is too high. Stop evacuation!
	// Set error
	M_SetError('Prevacuum pressure too high. Stopping evacuation...');
	ctrl.bEnable_Valve	:= FALSE;
	stat.nState			:= E_CRYO_EVAC_STATE.CLOSE_INSULATION_VALVE;	// Next state
	M_SetLabels();
END_IF
END_METHOD

METHOD M_Activity_Off
VAR_INPUT
END_VAR
// Disable anything that is not safe in this state
ctrl.bEnable_RP		:= FALSE;
ctrl.bEnable_TP		:= FALSE;
ctrl.bEnable_Valve	:= FALSE;


// System is started by setting in_bEnable to TRUE
trig(CLK := in_bEnable);

IF trig.Q THEN
	// Clear any existing error
	M_SetError('OK');
	
	// Enable Roughing Pump
	ctrl.bEnable_RP	:= TRUE;
	
	stat.nState	:= E_CRYO_EVAC_STATE.START_R_PUMP;	// Next state
	M_SetLabels();
END_IF
END_METHOD

METHOD M_Activity_OpeningValve
VAR_INPUT
END_VAR
IF NOT in_bEnable THEN
	// If system is disabled, start stopping procedure.
	ctrl.bEnable_Valve	:= FALSE;
	stat.nState			:= E_CRYO_EVAC_STATE.CLOSE_INSULATION_VALVE;	// Next state
	M_SetLabels();
ELSIF valve.stat.bActON THEN
	// The valve is open.
	// If valve was open before starting Turbo pump, 
	// wait for cryo pressure drop and then start the pump.
	// If the turbo pump is already running, the evacuation has started.
	IF NOT stat.bValveAfterTP	THEN
		stat.nState	:= E_CRYO_EVAC_STATE.WAIT_CRYO_VAC;	// Next state
	ELSE
		stat.nState	:= E_CRYO_EVAC_STATE.EVACUATING;	// Next state
	END_IF
	M_SetLabels();
END_IF
END_METHOD

METHOD M_Activity_StartingRoughingPump
VAR_INPUT
END_VAR
// Disable anything that is not safe in this state
ctrl.bEnable_TP		:= FALSE;
ctrl.bEnable_Valve	:= FALSE;


IF NOT in_bEnable THEN
	// If system is disabled, start stopping procedure.
	ctrl.bEnable_Valve	:= FALSE;
	stat.nState	:= E_CRYO_EVAC_STATE.CLOSE_INSULATION_VALVE;	// Next state
	M_SetLabels();
ELSIF rpRef.M_IsReady() THEN
	// Roughing Pump is Ready.
	// Wait for the prevacuum.
	stat.nState	:= E_CRYO_EVAC_STATE.WAIT_PREVAC;	// Next state
	M_SetLabels();
END_IF
END_METHOD

METHOD M_Activity_StartingTurboPump
VAR_INPUT
END_VAR
// Safety
// If the valve should be open after Turbo Pump has started,
// keep the valve closed.
IF stat.bValveAfterTP THEN
	ctrl.bEnable_Valve	:= FALSE;
END_IF

IF NOT in_bEnable THEN
	// If system is disabled, start stopping procedure.
	ctrl.bEnable_Valve	:= FALSE;
	stat.nState			:= E_CRYO_EVAC_STATE.CLOSE_INSULATION_VALVE;	// Next state
	M_SetLabels();
ELSIF tpRef.M_IsReady() THEN
	// Turbo Molecular Pump is Ready.
	// If the valve is not open, open it.
	// Otherwise, evacuation has started.
	IF stat.bValveAfterTP THEN
		ctrl.bEnable_Valve	:= TRUE;
		stat.nState			:= E_CRYO_EVAC_STATE.OPEN_INSULATION_VALVE;	// Next state
	ELSE
		stat.nState	:= E_CRYO_EVAC_STATE.EVACUATING;	// Next state
	END_IF
	M_SetLabels();
END_IF
END_METHOD

METHOD M_Activity_StoppingRoughingPump
VAR_INPUT
END_VAR
// Disable anything that is not safe in this state
ctrl.bEnable_RP		:= FALSE;
ctrl.bEnable_TP		:= FALSE;
ctrl.bEnable_Valve	:= FALSE;


// The evacuation system is in the process of shutting down.
// Allow re-starting of evacuation.
// System is started by setting in_bEnable to TRUE.
trig(CLK := in_bEnable);

IF trig.Q THEN
	// Clear any existing error
	M_SetError('OK');
	
	// Enable Roughing Pump
	ctrl.bEnable_RP	:= TRUE;
	
	stat.nState	:= E_CRYO_EVAC_STATE.START_R_PUMP;	// Next state
	M_SetLabels();
ELSIF NOT rpRef.M_IsRunning() THEN
	// The Roughing Pump stopped.
	// Wait for the Turbo Pump to get to complete stop.
	stat.nState	:= E_CRYO_EVAC_STATE.WAIT_T_PUMP_STOP;	// Next state
	M_SetLabels();
END_IF
END_METHOD

METHOD M_Activity_StoppingTurboPump
VAR_INPUT
END_VAR
// Disable anything that is not safe in this state
ctrl.bEnable_Valve	:= FALSE;


// The evacuation system is in the process of shutting down.
// Allow re-starting of evacuation.
// System is started by setting in_bEnable to TRUE.
trig(CLK := in_bEnable);

IF trig.Q THEN
	// Clear any existing error
	M_SetError('OK');
	
	// Enable Roughing Pump
	ctrl.bEnable_RP	:= TRUE;
	
	stat.nState	:= E_CRYO_EVAC_STATE.START_R_PUMP;	// Next state
	M_SetLabels();
ELSIF tpRef.M_GetSpeed() < 100 THEN
	// TODO: This is ATH2303M specific.
	//       Maybe, speed < 100 or similar check.
	
	// The Turbo Pump speed dropped below 100 rpm.
	// Stop the Roughing Pump.
	ctrl.bEnable_RP	:= FALSE;
	stat.nState		:= E_CRYO_EVAC_STATE.STOP_R_PUMP;	// Next state
	M_SetLabels();
END_IF
END_METHOD

METHOD M_Activity_WaitingCryoVacuum
VAR_INPUT
END_VAR
// Safety
// Disable Turbo Pump until it is safe to start.
ctrl.bEnable_TP	:= FALSE;

IF NOT in_bEnable THEN
	// If system is disabled, start stopping procedure.
	ctrl.bEnable_Valve	:= FALSE;
	stat.nState			:= E_CRYO_EVAC_STATE.CLOSE_INSULATION_VALVE;	// Next state
	M_SetLabels();
ELSIF in_lrCryoPressure <= cfg.lrThld_Valve_SafeOpenPressure THEN
	ctrl.bEnable_TP	:= TRUE;	// Enable Turbo Pump
	stat.nState		:= E_CRYO_EVAC_STATE.START_T_PUMP;	// Next state
	M_SetLabels();
END_IF
END_METHOD

METHOD M_Activity_WaitingPrevacuum
VAR_INPUT
END_VAR
// Disable anything that is not safe in this state
ctrl.bEnable_TP		:= FALSE;
ctrl.bEnable_Valve	:= FALSE;


IF NOT in_bEnable THEN
	// If system is disabled, start stopping procedure.
	ctrl.bEnable_Valve	:= FALSE;
	stat.nState	:= E_CRYO_EVAC_STATE.CLOSE_INSULATION_VALVE;	// Next state
	M_SetLabels();
ELSIF prevac.stat.lrPressure <= cfg.lrThld_Prevac THEN
	// If cryostat pressure is <= lrThldTP_SafeStartPressure, 
	// start Turbo Pump before opening the Insulation Valve.
	// Otherwise, open the Insulation Valve first.
	IF in_lrCryoPressure <= cfg.lrThld_TP_SafeStartPressure	THEN
		ctrl.bEnable_TP		:= TRUE;	// Enable Turbo Pump
		stat.bValveAfterTP	:= TRUE;	// Open valve after Turbo Pump has started
		stat.nState		:= E_CRYO_EVAC_STATE.START_T_PUMP;	// Next state
	ELSE
		ctrl.bEnable_Valve	:= TRUE;	// Open Valve
		stat.bValveAfterTP	:= FALSE;	// Valve opens before Turbo Pump starts
		stat.nState			:= E_CRYO_EVAC_STATE.OPEN_INSULATION_VALVE;	// Next state
	END_IF
	M_SetLabels();
END_IF
END_METHOD

METHOD M_Activity_WaitingTurboPump2Stop
VAR_INPUT
END_VAR
// Disable anything that is not safe in this state
ctrl.bEnable_RP		:= FALSE;
ctrl.bEnable_TP		:= FALSE;
ctrl.bEnable_Valve	:= FALSE;


// The evacuation system is in the process of shutting down.
// Allow re-starting of evacuation.
// System is started by setting in_bEnable to TRUE.
trig(CLK := in_bEnable);

IF trig.Q THEN
	// Clear any existing error
	M_SetError('OK');
	
	// Enable Roughing Pump
	ctrl.bEnable_RP	:= TRUE;
	
	stat.nState	:= E_CRYO_EVAC_STATE.START_R_PUMP;	// Next state
	M_SetLabels();
ELSIF tpRef.M_GetSpeed() = 0 THEN
	// The Turbo Pump came to complete stop.
	// The Evacuation system is OFF.
	stat.nState	:= E_CRYO_EVAC_STATE.OFF;	// Next state
	M_SetLabels();
END_IF
END_METHOD

METHOD M_Configure
VAR_INPUT
END_VAR
//
// TODO USER: If needed, overload this method with specific values.
//            This is the default configuration.
//
IF NOT stat.bConfigured	THEN
	// Specific instance configuration, e.g. anything different
	// from the default values given in the cfg structure of type T_CRYO_EVAC_CFG.
	cfg.nPressGaugeType1	:= E_CRYO_SENSOR_TYPE_PRESS.PKR_360;
	cfg.nPressGaugeType2	:= E_CRYO_SENSOR_TYPE_PRESS.PKR_360;

	cfg.lrThld_Prevac := 5.0;	// Prevacuum pressure threshold 5 mbar
	// Cryo pressure threshold to start Turbo Pump before opening Valve 10e-2 mbar
	cfg.lrThld_TP_SafeStartPressure := 0.01;	 
	// Cryo pressure threshold to start Turbo Pump once Valve is open 10e-1 mbar
	cfg.lrThld_Valve_SafeOpenPressure := 0.1;	
	cfg.tDelay := T#3S;	// Time delay before stopping Turbo Pump

	stat.bConfigured	:= TRUE;;
ELSE
	RETURN;	// Nothing to do any more
END_IF
END_METHOD

METHOD M_ExecuteControllers
VAR_INPUT
END_VAR
END_METHOD

METHOD M_GotoOff
VAR_INPUT
END_VAR
ctrl.bEnable_TP		:= FALSE;
ctrl.bEnable_RP		:= FALSE;
ctrl.bEnable_Valve	:= FALSE;
stat.nState			:= E_CRYO_EVAC_STATE.OFF;	// Next state
M_SetLabels();
END_METHOD

METHOD M_ReadSensors
VAR_INPUT
END_VAR
// Read prevacuum pressure sensors.
// Note: Pressure sensor type is configured in cfg.
//       Default is Pfeiffer PKR 360 KF25.
press1(in_nType := cfg.nPressGaugeType1, in_nSampleTime := 100);
press2(in_nType := cfg.nPressGaugeType2, in_nSampleTime := 100);
prevac(
	in_bSimulation	:= cfg.bPressSimulation,
	in_nNumSensor	:= 2,
	in_nVoteMethod	:= E_CRYO_VOTE.V_1oo2,
	in_pSensor1		:= ADR(press1),
	in_pSensor2		:= ADR(press2));
END_METHOD

METHOD M_SetError
VAR_INPUT
	in_sErrorText:	STRING(64);
END_VAR
stat.bError		:= (in_sErrorText <> 'OK');
stat.sErrorText	:= in_sErrorText;
END_METHOD

METHOD M_SetLabels
VAR_INPUT
END_VAR
VAR
    fbFormat:	FB_FormatString;
	nVal:		UDINT;
	lrVal:		LREAL;
END_VAR
CASE stat.nState	OF
	E_CRYO_EVAC_STATE.NONE:
		stat.sState		:= 'NONE';
		stat.sStatus	:= 'UNKNOWN';
	E_CRYO_EVAC_STATE.OFF:
		stat.sState		:= 'OFF';
		stat.sStatus	:= 'OFF';
	E_CRYO_EVAC_STATE.START_R_PUMP:
		stat.sState		:= 'START_R_PUMP';
		stat.sStatus	:= 'Starting Roughing Pump...';
	E_CRYO_EVAC_STATE.WAIT_PREVAC:
		stat.sState		:= 'WAIT_PREVAC';
		fbFormat(	sFormat := 'Waiting Prevacuum Pressure <= %.4f [mbar]...', 
					arg1 := F_LREAL(cfg.lrThld_Prevac), 
					sOut => stat.sStatus);
	E_CRYO_EVAC_STATE.OPEN_INSULATION_VALVE:
		stat.sState		:= 'OPEN_INSULATION_VALVE';
		stat.sStatus	:= 'Opening Insulation Valve...';
	E_CRYO_EVAC_STATE.START_T_PUMP:
		stat.sState		:= 'START_T_PUMP';
		stat.sStatus	:= 'Starting Turbo Molecular Pump...';
	E_CRYO_EVAC_STATE.WAIT_CRYO_VAC:
		stat.sState		:= 'WAIT_CRYO_VAC';
		// The target cryostat pressure depends on whether the valve is open or not.
		IF valve.stat.bActON THEN
			lrVal	:= cfg.lrThld_Valve_SafeOpenPressure;
		ELSE
			lrVal	:= cfg.lrThld_TP_SafeStartPressure;
		END_IF
		fbFormat(	sFormat := 'Waiting Cryostat Pressure <= %.4f [mbar]...', 
					arg1 := F_LREAL(lrVal), 
					sOut => stat.sStatus);
	E_CRYO_EVAC_STATE.EVACUATING:
		stat.sState		:= 'EVACUATING';
		stat.sStatus	:= 'EVACUATING...';
	E_CRYO_EVAC_STATE.CLOSE_INSULATION_VALVE:
		stat.sState		:= 'CLOSE_INSULATION_VALVE';
		stat.sStatus	:= 'Closing Insulation Valve...';
	E_CRYO_EVAC_STATE.DELAY_STOPPING:
		stat.sState		:= 'DELAY_STOPPING';
		nVal			:= TIME_TO_UDINT(cfg.tDelay);
		fbFormat(	sFormat := 'Delay of %d [ms] Before Stopping Pumps...', 
					arg1 := F_UDINT(nVal), 
					sOut => stat.sStatus);
	E_CRYO_EVAC_STATE.STOP_T_PUMP:
		stat.sState		:= 'STOP_T_PUMP';
		stat.sStatus	:= 'Stopping Turbo Molecular Pump...';
	E_CRYO_EVAC_STATE.STOP_R_PUMP:
		stat.sState		:= 'STOP_R_PUMP';
		stat.sStatus	:= 'Stopping Roughing Pump...';
	E_CRYO_EVAC_STATE.WAIT_T_PUMP_STOP:
		stat.sState		:= 'WAIT_T_PUMP_STOP';
		stat.sStatus	:= 'Waiting for Turbo Molecular Pump to Stop...';
	
END_CASE
END_METHOD

METHOD M_StateMachine
VAR_INPUT
END_VAR
CASE stat.nState	OF
	E_CRYO_EVAC_STATE.NONE:
		M_GotoOff();
	E_CRYO_EVAC_STATE.OFF:
		M_Activity_Off();
	E_CRYO_EVAC_STATE.START_R_PUMP:
		M_Activity_StartingRoughingPump();
	E_CRYO_EVAC_STATE.WAIT_PREVAC:
		M_Activity_WaitingPrevacuum();
	E_CRYO_EVAC_STATE.OPEN_INSULATION_VALVE:
		M_Activity_OpeningValve();
	E_CRYO_EVAC_STATE.START_T_PUMP:
		M_Activity_StartingTurboPump();
	E_CRYO_EVAC_STATE.WAIT_CRYO_VAC:
		M_Activity_WaitingCryoVacuum();
	E_CRYO_EVAC_STATE.EVACUATING:
		M_Activity_Evacuating();
	E_CRYO_EVAC_STATE.CLOSE_INSULATION_VALVE:
		M_Activity_ClosingValve();
	E_CRYO_EVAC_STATE.DELAY_STOPPING:
		M_Activity_DelayBeforeStoppingPumps();
	E_CRYO_EVAC_STATE.STOP_T_PUMP:
		M_Activity_StoppingTurboPump();
	E_CRYO_EVAC_STATE.STOP_R_PUMP:
		M_Activity_StoppingRoughingPump();
	E_CRYO_EVAC_STATE.WAIT_T_PUMP_STOP:
		M_Activity_WaitingTurboPump2Stop();
	
END_CASE
END_METHOD

METHOD M_UpdateStatus
VAR_INPUT
END_VAR
stat.bEnabled		:= in_bEnable;
stat.bRootPumpON	:= rpRef.M_IsReady();
stat.bTurboPumpON	:= tpRef.M_IsReady();
stat.bValveOpen		:= valve.stat.bActON;
END_METHOD

END_FUNCTION_BLOCK

// POUs/Subsystems/Evacuation/FB_CRYO_EVAC_BASE_50000
FUNCTION_BLOCK FB_CRYO_EVAC_BASE_50000
VAR_INPUT
	in_bEnable:		BOOL := FALSE;	// System active while in_bEnable is TRUE
	in_RefVAGF:		REFERENCE TO FB_CRYO_PRESSURE_VOTE;
	in_RefVAGG:		REFERENCE TO FB_CRYO_PRESSURE_VOTE;
END_VAR
VAR_OUTPUT
END_VAR
VAR
	/////////
	// Pumps
	/////////
	
	rpRef:	REFERENCE TO FB_CRYO_PUMP_BASE;		// Roughing Pump
	tpRef:	REFERENCE TO FB_CRYO_PUMP_BASE;		// Turbo Molecular Pump
	
	//////////
	// Valves
	//////////
	
	PVV1:	FB_CRYO_VALVE_CTRL;					// Prevacuum Valve #1
	PVV2:	FB_CRYO_VALVE_CTRL;					// Prevacuum Valve #2
	PVV3:	FB_CRYO_VALVE_CTRL;					// Prevacuum Valve #3
	PVV4:	FB_CRYO_VALVE_CTRL;					// Prevacuum Valve #4
	GBV:	FB_CRYO_VALVE_CTRL;					// Gas-ballast Valve
	
	// Valve command handling
	cmdPVV1:	FB_CRYO_ACTUATOR_CMD;
	cmdPVV2:	FB_CRYO_ACTUATOR_CMD;
	cmdPVV3:	FB_CRYO_ACTUATOR_CMD;
	cmdPVV4:	FB_CRYO_ACTUATOR_CMD;
	cmdGBV:		FB_CRYO_ACTUATOR_CMD;

	
	// Pointers to valves
	ptrV:	ARRAY [1..5] OF POINTER TO FB_CRYO_VALVE_CTRL;
	// Pointers to valve commands
	ptrVC:	ARRAY [1..5] OF POINTER TO FB_CRYO_ACTUATOR_CMD;
	// Pointers to Enable flags for valves
	ptrEV:	ARRAY [1..5] OF POINTER TO BOOL;
	
	////////////
	// Pressure
	////////////
	
	// Pressure transducers
	sensor_VAG1:	FB_CRYO_SENSOR_PRESSURE;	// Prevacuum pressure gauge #1
	sensor_VAG2:	FB_CRYO_SENSOR_PRESSURE;	// Prevacuum pressure gauge #2
	sensor_VAG3:	FB_CRYO_SENSOR_PRESSURE;	// Prevacuum pressure gauge #3

	
	// Pressure measurements
	VAG1:	FB_CRYO_PRESSURE_VOTE;				// Prevacuum pressure #1
	VAG2:	FB_CRYO_PRESSURE_VOTE;				// Prevacuum pressure #2
	VAG3:	FB_CRYO_PRESSURE_VOTE;				// Prevacuum pressure #3
	VAGF:	FB_CRYO_PRESSURE_VOTE;				// Cryo pressure F
	VAGG:	FB_CRYO_PRESSURE_VOTE;				// Cryo pressure G
	// Pointers to pressures
	ptrP:	ARRAY [1..5] OF POINTER TO FB_CRYO_PRESSURE_VOTE;
	
	
	cfg:	T_CRYO_EVAC_CFG_50000;
	ctrl:	T_CRYO_EVAC_CTRL_50000;
	stat:	T_CRYO_EVAC_STAT_50000;
	
	timer:	TON;
	trig:	R_TRIG;	// Start trigger
	
	// GUI staff
	guiValveIndex:	UINT := 1;	// Index for Valve Engineering GUI
END_VAR

// NOTE: Configuration is set on the first cycle.
//       Once stat.bConfigured is TRUE, 
//       configuration is not updated any more.
M_Configure();

M_ReadSensors();

M_ExecuteControllers();

M_UpdateStatus();

M_StateMachine();

METHOD M_ActionExecute
VAR_INPUT
END_VAR
CASE stat.nState	OF
	E_CRYO_EVAC_STATE_50000.NONE:
		;	// Nothing to do

	E_CRYO_EVAC_STATE_50000.OFF:
		;	// Nothing to do

	E_CRYO_EVAC_STATE_50000.START_PVP:
		ctrl.bEnable_PVP	:= TRUE;
		ctrl.bEnable_PVV1	:= FALSE;
		ctrl.bEnable_PVV2	:= FALSE;
		ctrl.bEnable_PVV3	:= FALSE;
		ctrl.bEnable_PVV4	:= FALSE;
		ctrl.bEnable_GBV	:= FALSE;

	E_CRYO_EVAC_STATE_50000.OPEN_GBV:
		ctrl.bEnable_GBV	:= TRUE;

	E_CRYO_EVAC_STATE_50000.WAIT_VAG3:
		;	// Nothing to do

	E_CRYO_EVAC_STATE_50000.OPEN_PVV1:
		ctrl.bEnable_PVV1	:= TRUE;

	E_CRYO_EVAC_STATE_50000.WAIT_VAG_1_3:
		;	// Nothing to do

	E_CRYO_EVAC_STATE_50000.OPEN_PVV2:
		ctrl.bEnable_PVV2	:= TRUE;

	E_CRYO_EVAC_STATE_50000.WAIT_VAG_F_G_1:
		;	// Nothing to do

	E_CRYO_EVAC_STATE_50000.CLOSE_PVV2:
		ctrl.bEnable_PVV2	:= FALSE;

	E_CRYO_EVAC_STATE_50000.CLOSE_PVV1:
		ctrl.bEnable_PVV1	:= FALSE;

	E_CRYO_EVAC_STATE_50000.START_TMP:
		ctrl.bEnable_TMP	:= TRUE;
		
	E_CRYO_EVAC_STATE_50000.OPEN_PVV3:
		ctrl.bEnable_PVV3	:= TRUE;

	E_CRYO_EVAC_STATE_50000.WAIT_VAG_2_3:
		;	// Nothing to do

	E_CRYO_EVAC_STATE_50000.OPEN_PVV4:
		ctrl.bEnable_PVV4	:= TRUE;

	E_CRYO_EVAC_STATE_50000.WAIT_VAG_F_G_2:
		;	// Nothing to do

	E_CRYO_EVAC_STATE_50000.CLOSE_GBV:
		ctrl.bEnable_GBV	:= FALSE;

	E_CRYO_EVAC_STATE_50000.EVACUATING:
		;	// Nothing to do

	E_CRYO_EVAC_STATE_50000.CLOSE_ALL_VALVES:
		ctrl.bEnable_PVV1	:= FALSE;
		ctrl.bEnable_PVV2	:= FALSE;
		ctrl.bEnable_PVV3	:= FALSE;
		ctrl.bEnable_PVV4	:= FALSE;
		ctrl.bEnable_GBV	:= FALSE;

	E_CRYO_EVAC_STATE_50000.DELAY_STOPPING:
		;	// Nothing to do

	E_CRYO_EVAC_STATE_50000.STOP_TMP_1:
		ctrl.bEnable_TMP	:= FALSE;

	E_CRYO_EVAC_STATE_50000.STOP_PVP:
		ctrl.bEnable_PVP	:= FALSE;

	E_CRYO_EVAC_STATE_50000.WAIT_TMP_STANDSTILL:
		;	// Nothing to do

	E_CRYO_EVAC_STATE_50000.STOP_TMP_2:
		ctrl.bEnable_TMP	:= FALSE;
	
END_CASE

timer(IN:=FALSE);	// Reset timer, just in case.
END_METHOD

METHOD M_Activity_ClosingAllValves
VAR_INPUT
END_VAR
VAR
	i:			INT;
	bAllClosed:	BOOL := TRUE;
END_VAR
// Check all valves if they are closed.
// If any of them is not closed, then they are not all closed.
FOR i := 1 TO 5 DO
	IF NOT ptrV[i]^.stat.bActOFF	THEN
		bAllClosed	:= FALSE;
		EXIT;
	END_IF
END_FOR

IF bAllClosed THEN
	// All valves are closed.
	// In next state apply a delay before stopping pumps.
	M_SetNextState(E_CRYO_EVAC_STATE_50000.DELAY_STOPPING);
END_IF
END_METHOD

METHOD M_Activity_ClosingValve
VAR_INPUT
	index:		INT;
	nNextState:	E_CRYO_EVAC_STATE_50000;	// Next state after valve is closed
END_VAR
// Check if valve index is valid.
// If not, just return (for safety).
IF index < 1  OR  index > 5	THEN
	RETURN;
END_IF 

IF ptrV[index]^.stat.bActOFF THEN
	// The valve is closed.
	// Set next state and execute its action
	M_SetNextState(nNextState);	// Next state
	
END_IF
END_METHOD

METHOD M_Activity_DelayBeforeStoppingPumps
VAR_INPUT
END_VAR
timer(IN:=TRUE, PT:=CFG.tDelay);

IF timer.Q THEN
	// Delay timer expired.
	// Reset timer.
	timer(IN:=FALSE);
	
	// Stop Turbo Pump.
	M_SetNextState(E_CRYO_EVAC_STATE_50000.STOP_TMP_1);	// Next state

END_IF
END_METHOD

METHOD M_Activity_Evacuating
VAR_INPUT
END_VAR
VAR
	index1:	INT	:= E_CRYO_EVAC_PRESSURES_50000.VAG2;
	index2:	INT	:= E_CRYO_EVAC_PRESSURES_50000.VAG3;
END_VAR
// System is started by setting in_bEnable to TRUE
IF NOT in_bEnable THEN
	// If system is disabled, start stopping procedure.
	M_SetNextState(E_CRYO_EVAC_STATE_50000.CLOSE_ALL_VALVES);	// Next state
	
ELSIF 	ptrP[index1]^.stat.lrPressure > cfg.lrThld_PrevacHigh  AND
		ptrP[index2]^.stat.lrPressure > cfg.lrThld_PrevacHigh THEN
	// Something is wrong. Prevacuum pressure is too high. Stop evacuation!
	// Set error.
	M_SetError('Prevacuum pressure too high. Stopping evacuation...');
	M_SetNextState(E_CRYO_EVAC_STATE_50000.CLOSE_ALL_VALVES);	// Next state
	
END_IF
END_METHOD

METHOD M_Activity_Off
VAR_INPUT
END_VAR
// Disable anything that is not safe in this state
ctrl.bEnable_PVP	:= FALSE;
ctrl.bEnable_TMP	:= FALSE;
ctrl.bEnable_PVV1	:= FALSE;
ctrl.bEnable_PVV2	:= FALSE;
ctrl.bEnable_PVV3	:= FALSE;
ctrl.bEnable_PVV4	:= FALSE;
ctrl.bEnable_GBV	:= FALSE;


// System is started by setting in_bEnable to TRUE
trig(CLK := in_bEnable);

IF trig.Q THEN
	// Clear any existing error
	M_SetError('OK');
	
	M_SetNextState(E_CRYO_EVAC_STATE_50000.START_PVP);	// Next state
END_IF
END_METHOD

METHOD M_Activity_OpeningValve
VAR_INPUT
	index:		INT;
	nNextState:	E_CRYO_EVAC_STATE_50000;	// Next state after valve is closed
END_VAR
IF NOT in_bEnable THEN
	// If system is disabled, start stopping procedure.
	M_SetNextState(E_CRYO_EVAC_STATE_50000.CLOSE_ALL_VALVES);	// Next state
	
ELSIF ptrV[index]^.stat.bActON THEN
	// The valve is open.
	// Go to next state
	M_SetNextState(nNextState);
	
END_IF
END_METHOD

METHOD M_Activity_StartingPVP
VAR_INPUT
END_VAR
// Disable anything that is not safe in this state
ctrl.bEnable_TMP	:= FALSE;
ctrl.bEnable_PVV1	:= FALSE;
ctrl.bEnable_PVV2	:= FALSE;
ctrl.bEnable_PVV3	:= FALSE;
ctrl.bEnable_PVV4	:= FALSE;
ctrl.bEnable_GBV	:= FALSE;


IF NOT in_bEnable THEN
	// If system is disabled, start stopping procedure.
	M_SetNextState(E_CRYO_EVAC_STATE_50000.CLOSE_ALL_VALVES);	// Next state
	
ELSIF rpRef.M_IsReady() THEN
	// Roughing Pump is Ready.
	// Open Gas-ballast valve.
	M_SetNextState(E_CRYO_EVAC_STATE_50000.OPEN_GBV);	// Next state
	
END_IF
END_METHOD

METHOD M_Activity_StartingTMP
VAR_INPUT
END_VAR
VAR
	index1:	INT	:= E_CRYO_EVAC_PRESSURES_50000.VAGF;
	index2:	INT	:= E_CRYO_EVAC_PRESSURES_50000.VAGG;
END_VAR
IF NOT in_bEnable THEN
	// If system is disabled, start stopping procedure by closing all valves.
	M_SetNextState(E_CRYO_EVAC_STATE_50000.CLOSE_ALL_VALVES);	// Next state
	
ELSIF 	ptrP[index1]^.stat.lrPressure > cfg.lrThld_Prevac  OR
		ptrP[index2]^.stat.lrPressure > cfg.lrThld_Prevac 	THEN
	// Cryostat pressure is too high for some reason.
	// Stop Turbo Molecular pump.
	M_SetNextState(E_CRYO_EVAC_STATE_50000.STOP_TMP_2);
		
ELSIF tpRef.M_IsReady() THEN
	// Turbo Molecular Pump is Ready, i.e., running at operational speed.
	// Open PVV3.
	M_SetNextState(E_CRYO_EVAC_STATE_50000.OPEN_PVV3);	// Next state
	
END_IF
END_METHOD

METHOD M_Activity_StoppingPVP
VAR_INPUT
END_VAR
// Disable anything that is not safe in this state
ctrl.bEnable_PVP	:= FALSE;
ctrl.bEnable_TMP	:= FALSE;


// The evacuation system is in the process of shutting down.
// Allow re-starting of evacuation.
// System is started by setting in_bEnable to TRUE.
trig(CLK := in_bEnable);

IF trig.Q THEN
	// Clear any existing error
	M_SetError('OK');
	
	// Enable Roughing Pump
	M_SetNextState(E_CRYO_EVAC_STATE_50000.START_PVP);
	
ELSIF NOT rpRef.M_IsRunning() THEN
	// The Roughing Pump stopped.
	// Wait for the Turbo Pump to get to complete stop.
	M_SetNextState(E_CRYO_EVAC_STATE_50000.WAIT_TMP_STANDSTILL);	// Next state

END_IF
END_METHOD

METHOD M_Activity_StoppingTMP
VAR_INPUT
	index:	INT;	// Index of action(1 or 2, for STP_TMP and STOP2_TMP)
END_VAR
// Disable anything that is not safe in this state


// The evacuation system is in the process of shutting down.
// Allow re-starting of evacuation.
// System is started by setting in_bEnable to TRUE.
trig(CLK := in_bEnable);

IF trig.Q THEN
	// Clear any existing error
	M_SetError('OK');
	
	// Enable Roughing Pump
	M_SetNextState(E_CRYO_EVAC_STATE_50000.START_PVP);
	
ELSIF NOT tpRef.M_IsReady() THEN
	// TODO: This is ATH2303M specific.
	//       Maybe, speed < 100 or similar check.
	
	IF index = 1	THEN
		// Case 1: Proceed with stopping PVP.
		M_SetNextState(E_CRYO_EVAC_STATE_50000.STOP_PVP);
	ELSIF index = 2	THEN
		// Case 2: Proceed with openning PVV1.
		M_SetNextState(E_CRYO_EVAC_STATE_50000.OPEN_PVV1);
	END_IF
	
END_IF
END_METHOD

METHOD M_Activity_Waiting2Pressures
VAR_INPUT
	index1:		INT;
	index2:		INT;
	lrRef:		LREAL;	// Reference pressure [mbar]
	nNextState:	E_CRYO_EVAC_STATE_50000;	// Next state after pressure is reached
END_VAR
// Check if valve indexes are valid. Range [1..5]
// If not, just return (for safety).
IF index1 < 1  OR  index1 > 5  OR  index2 < 1  OR  index2 > 5  THEN
	RETURN;
END_IF 

IF	(ptrP[index1]^.stat.bValid  AND  ptrP[index1]^.stat.lrPressure < lrRef)  AND
	(ptrP[index2]^.stat.bValid  AND  ptrP[index2]^.stat.lrPressure < lrRef)  	THEN
	// The pressure has been reached.
	
	M_SetNextState(nNextState);	// Next state
END_IF
END_METHOD

METHOD M_Activity_WaitingPressure
VAR_INPUT
	index:		INT;
	lrRef:		LREAL;	// Reference pressure [mbar]
	nNextState:	E_CRYO_EVAC_STATE_50000;	// Next state after pressure is reached
END_VAR
// Check if valve index is valid.
// If not, just return (for safety).
IF index < 1  OR  index > 5	THEN
	RETURN;
END_IF 

IF ptrP[index]^.stat.bValid  AND  ptrP[index]^.stat.lrPressure < lrRef  THEN
	// The pressure has been reached.
	
	M_SetNextState(nNextState);	// Next state
END_IF
END_METHOD

METHOD M_Activity_WaitingTMP2Stop
VAR_INPUT
END_VAR
// Disable anything that is not safe in this state
ctrl.bEnable_PVP	:= FALSE;
ctrl.bEnable_TMP	:= FALSE;


// The evacuation system is in the process of shutting down.
// Allow re-starting of evacuation.
// System is started by setting in_bEnable to TRUE.
trig(CLK := in_bEnable);

IF trig.Q THEN
	// Clear any existing error
	M_SetError('OK');
	
	// Enable Roughing Pump
	M_SetNextState(E_CRYO_EVAC_STATE_50000.START_PVP);
	
ELSIF tpRef.M_GetSpeed() = 0 THEN
	// The Turbo Pump came to complete stop.
	// The Evacuation system is OFF.
	M_SetNextState(E_CRYO_EVAC_STATE_50000.OFF);
	
END_IF
END_METHOD

METHOD M_Configure
VAR_INPUT
END_VAR
//
// TODO USER: 
// This M_Configure() MUST be called once in the child FB M_Configure() method!!!
// It sets all the pointers to various variables.
// 
(*
//
// TODO USER in child FB
//
	// MANDATORY: Set References to pumps!!!
	// If not done, system will crash !!!
	rpRef	REF=rp;
	tpRef	REF=tp;
	
	// Specific instance configuration, e.g. pressure gauges' types.
	// See FB_CRYO_EVAC_MICADO::M_Configure().
	// ...

*)	

// Set pointers to Valves - MUST!!!
ptrV[1]	:= ADR(PVV1);
ptrV[2]	:= ADR(PVV2);
ptrV[3]	:= ADR(PVV3);
ptrV[4]	:= ADR(PVV4);
ptrV[5]	:= ADR(GBV);

// Set pointers to Valve Commands - MUST!!!
ptrVC[1]	:= ADR(cmdPVV1);
ptrVC[2]	:= ADR(cmdPVV2);
ptrVC[3]	:= ADR(cmdPVV3);
ptrVC[4]	:= ADR(cmdPVV4);
ptrVC[5]	:= ADR(cmdGBV);

// Set pointers to Enable Valves flags - MUST!!!
ptrEV[1]	:= ADR(ctrl.bEnable_PVV1);
ptrEV[2]	:= ADR(ctrl.bEnable_PVV2);
ptrEV[3]	:= ADR(ctrl.bEnable_PVV3);
ptrEV[4]	:= ADR(ctrl.bEnable_PVV4);
ptrEV[5]	:= ADR(ctrl.bEnable_GBV);


// Set pointers to Pressures - MUST!!!
ptrP[1]	:= ADR(VAG1);
ptrP[2]	:= ADR(VAG2);
ptrP[3]	:= ADR(VAG3);
ptrP[4]	:= ADR(VAGF);
ptrP[5]	:= ADR(VAGG);
END_METHOD

METHOD M_ExecuteControllers
VAR_INPUT
END_VAR
// Valve commands
cmdPVV1(in_bEnable := ctrl.bEnable_PVV1);	// Handling of PVV1 commands
cmdPVV2(in_bEnable := ctrl.bEnable_PVV2);	// Handling of PVV2 commands
cmdPVV3(in_bEnable := ctrl.bEnable_PVV3);	// Handling of PVV3 commands
cmdPVV4(in_bEnable := ctrl.bEnable_PVV4);	// Handling of PVV4 commands
cmdGBV (in_bEnable := ctrl.bEnable_GBV);	// Handling of GBV  commands

// Valve Control
PVV1(
	in_bEnable			:= cmdPVV1.out_bEnable,
	in_nFeedback		:= E_CRYO_BIN_ACT_FEEDBACK.ON_AND_OFF);

PVV2(
	in_bEnable			:= cmdPVV2.out_bEnable,
	in_nFeedback		:= E_CRYO_BIN_ACT_FEEDBACK.ON_AND_OFF);

PVV3(
	in_bEnable			:= cmdPVV3.out_bEnable,
	in_nFeedback		:= E_CRYO_BIN_ACT_FEEDBACK.ON_AND_OFF);

PVV4(
	in_bEnable			:= cmdPVV4.out_bEnable,
	in_nFeedback		:= E_CRYO_BIN_ACT_FEEDBACK.ON_AND_OFF);

GBV(
	in_bEnable			:= cmdGBV.out_bEnable,
	in_nFeedback		:= E_CRYO_BIN_ACT_FEEDBACK.ON_AND_OFF);
END_METHOD

METHOD M_ReadSensors
VAR_INPUT
END_VAR
///////////////////////////////////////////////
// Read individual prevacuum pressure sensors.
///////////////////////////////////////////////
//
// Pressure readings are averaged over 100 ms.
//
// Note: Pressure sensor type is configured in cfg and overwritten in M_Configure().
//       Default is Pfeiffer PKR 360 KF25.
sensor_VAG1	(in_nType := cfg.nType_VAG1,	in_nSampleTime := 100);
sensor_VAG2	(in_nType := cfg.nType_VAG2,	in_nSampleTime := 100);
sensor_VAG3	(in_nType := cfg.nType_VAG3,	in_nSampleTime := 100);
(*
sensor_VAGF1(in_nType := cfg.nType_VAGF1,	in_nSampleTime := 100);
sensor_VAGF2(in_nType := cfg.nType_VAGF2,	in_nSampleTime := 100);
sensor_VAGG1(in_nType := cfg.nType_VAGG1,	in_nSampleTime := 100);
sensor_VAGG2(in_nType := cfg.nType_VAGG2,	in_nSampleTime := 100);
*)

//////////////////////////////////////////////
// Use voting system to calculate pressures.
//////////////////////////////////////////////
//
// Note: VAG 1-3 have got only one sensor pressure connected !!!
//       VAG F & G have got two pressure sensors connected !
//
VAG1(
	in_bSimulation	:= cfg.bPressSimulation,
	in_nNumSensor	:= 2,
	in_nVoteMethod	:= E_CRYO_VOTE.V_1oo2,
	in_pSensor1		:= ADR(sensor_VAG1));

VAG2(
	in_bSimulation	:= cfg.bPressSimulation,
	in_nNumSensor	:= 2,
	in_nVoteMethod	:= E_CRYO_VOTE.V_1oo2,
	in_pSensor1		:= ADR(sensor_VAG2));

VAG3(
	in_bSimulation	:= cfg.bPressSimulation,
	in_nNumSensor	:= 2,
	in_nVoteMethod	:= E_CRYO_VOTE.V_1oo2,
	in_pSensor1		:= ADR(sensor_VAG3));

	
// Copy pressure references to local variables
VAGF	:= in_RefVAGF;
VAGG	:= in_RefVAGG;

	
(*	
VAGF(
	in_bSimulation	:= cfg.bPressSimulation,
	in_nNumSensor	:= 2,
	in_nVoteMethod	:= E_CRYO_VOTE.V_1oo2,
	in_pSensor1		:= ADR(sensor_VAGF1),
	in_pSensor2		:= ADR(sensor_VAGF2));

VAGG(
	in_bSimulation	:= cfg.bPressSimulation,
	in_nNumSensor	:= 2,
	in_nVoteMethod	:= E_CRYO_VOTE.V_1oo2,
	in_pSensor1		:= ADR(sensor_VAGG1),
	in_pSensor2		:= ADR(sensor_VAGG2));
*)
END_METHOD

METHOD M_SetError
VAR_INPUT
	in_sErrorText:	STRING(64);
END_VAR
stat.bError		:= (in_sErrorText <> 'OK');
stat.sErrorText	:= in_sErrorText;
END_METHOD

METHOD M_SetLabels
VAR_INPUT
END_VAR
VAR
    fbFormat:	FB_FormatString;
	nVal:		UDINT;
	lrVal:		LREAL;
END_VAR
CASE stat.nState	OF
	E_CRYO_EVAC_STATE_50000.NONE:
		stat.sState		:= 'NONE';
		stat.sStatus	:= 'UNKNOWN';
		
	E_CRYO_EVAC_STATE_50000.OFF:
		stat.sState		:= 'OFF';
		stat.sStatus	:= 'OFF';
		
	E_CRYO_EVAC_STATE_50000.START_PVP:
		stat.sState		:= 'START_PVP';
		stat.sStatus	:= 'Starting Roughing Pump...';
		
	E_CRYO_EVAC_STATE_50000.START_TMP:
		stat.sState		:= 'START_TMP';
		stat.sStatus	:= 'Starting Turbo Molecular Pump...';
		
	E_CRYO_EVAC_STATE_50000.STOP_TMP_1,
	E_CRYO_EVAC_STATE_50000.STOP_TMP_2:
		stat.sState		:= 'STOP_TMP_x';
		stat.sStatus	:= 'Stopping Turbo Molecular Pump...';
		
	E_CRYO_EVAC_STATE_50000.STOP_PVP:
		stat.sState		:= 'STOP_PVP';
		stat.sStatus	:= 'Stopping Roughing Pump...';
		
	E_CRYO_EVAC_STATE_50000.WAIT_VAG3:
		stat.sState		:= 'WAIT_VAG3';
		fbFormat(	sFormat := 'Waiting VAG3 <= %.4f [mbar]...', 
					arg1 := F_LREAL(cfg.lrThld_Prevac), 
					sOut => stat.sStatus);
					
	E_CRYO_EVAC_STATE_50000.WAIT_VAG_1_3:
		stat.sState		:= 'WAIT_VAG_1_3';
		fbFormat(	sFormat := 'Waiting VAG1 & VAG3 <= %.4f [mbar]...', 
					arg1 := F_LREAL(cfg.lrThld_Prevac), 
					sOut => stat.sStatus);
					
	E_CRYO_EVAC_STATE_50000.WAIT_VAG_2_3:
		stat.sState		:= 'WAIT_VAG_2_3';
		fbFormat(	sFormat := 'Waiting VAG2 & VAG3 <= %.4f [mbar]...', 
					arg1 := F_LREAL(cfg.lrThld_Prevac), 
					sOut => stat.sStatus);
					
	E_CRYO_EVAC_STATE_50000.WAIT_VAG_F_G_1:
		stat.sState		:= 'WAIT_VAG_F_G_1';
		lrVal			:= 0.9 * cfg.lrThld_Prevac;
		fbFormat(	sFormat := 'Waiting VAGF & VAGG <= %.4f [mbar]...', 
					arg1 := F_LREAL(lrVal), 
					sOut => stat.sStatus);
					
	E_CRYO_EVAC_STATE_50000.WAIT_VAG_F_G_2:
		stat.sState		:= 'WAIT_VAG_F_G_2';
		fbFormat(	sFormat := 'Waiting VAGF & VAGG <= %.4f [mbar]...', 
					arg1 := F_LREAL(cfg.lrThld_Vacuum), 
					sOut => stat.sStatus);
					
	E_CRYO_EVAC_STATE_50000.OPEN_PVV1:
		stat.sState		:= 'OPEN_PVV1';
		stat.sStatus	:= 'Opening PVV1 Valve...';

	E_CRYO_EVAC_STATE_50000.OPEN_PVV2:
		stat.sState		:= 'OPEN_PVV2';
		stat.sStatus	:= 'Opening PVV2 Valve...';

	E_CRYO_EVAC_STATE_50000.OPEN_PVV3:
		stat.sState		:= 'OPEN_PVV3';
		stat.sStatus	:= 'Opening PVV3 Valve...';

	E_CRYO_EVAC_STATE_50000.OPEN_PVV4:
		stat.sState		:= 'OPEN_PVV4';
		stat.sStatus	:= 'Opening PVV4 Valve...';
	
	E_CRYO_EVAC_STATE_50000.OPEN_GBV:
		stat.sState		:= 'OPEN_GBV';
		stat.sStatus	:= 'Opening Gas-ballast Valve...';

	E_CRYO_EVAC_STATE_50000.CLOSE_PVV1:
		stat.sState		:= 'CLOSE_PVV1';
		stat.sStatus	:= 'Closing PVV1 Valve...';

	E_CRYO_EVAC_STATE_50000.CLOSE_PVV2:
		stat.sState		:= 'CLOSE_PVV2';
		stat.sStatus	:= 'Closing PVV2 Valve...';

	E_CRYO_EVAC_STATE_50000.CLOSE_GBV:
		stat.sState		:= 'CLOSE_GBV';
		stat.sStatus	:= 'Closing GBV Valve...';

	E_CRYO_EVAC_STATE_50000.CLOSE_ALL_VALVES:
		stat.sState		:= 'CLOSE_ALL_VALVES';
		stat.sStatus	:= 'Closing All Valves...';
		
	E_CRYO_EVAC_STATE_50000.EVACUATING:
		stat.sState		:= 'EVACUATING';
		stat.sStatus	:= 'EVACUATING...';
		
	E_CRYO_EVAC_STATE_50000.DELAY_STOPPING:
		stat.sState		:= 'DELAY_STOPPING';
		nVal			:= TIME_TO_UDINT(cfg.tDelay);
		fbFormat(	sFormat := 'Delay of %d [ms] Before Stopping Pumps...', 
					arg1 := F_UDINT(nVal), 
					sOut => stat.sStatus);
					
	E_CRYO_EVAC_STATE_50000.WAIT_TMP_STANDSTILL:
		stat.sState		:= 'WAIT_TMP_STANDSTILL';
		stat.sStatus	:= 'Waiting for Turbo Molecular Pump to get Standstill...';
	
END_CASE
END_METHOD

METHOD M_SetNextState
VAR_INPUT
	nNextState:	E_CRYO_EVAC_STATE_50000;	// Next state
END_VAR
stat.nState	:= nNextState;	// Next state
M_ActionExecute();			// Execute Action for next state
M_SetLabels();
END_METHOD

METHOD M_StateMachine
VAR_INPUT
END_VAR
CASE stat.nState	OF
	E_CRYO_EVAC_STATE_50000.NONE:
		M_SetNextState(E_CRYO_EVAC_STATE_50000.OFF);
	E_CRYO_EVAC_STATE_50000.OFF:
		M_Activity_Off();

	E_CRYO_EVAC_STATE_50000.START_PVP:
		M_Activity_StartingPVP();

	E_CRYO_EVAC_STATE_50000.OPEN_GBV:
		M_Activity_OpeningValve(
			index		:= E_CRYO_EVAC_VALVES_50000.GBV, 
			nNextState	:= E_CRYO_EVAC_STATE_50000.WAIT_VAG3);

	E_CRYO_EVAC_STATE_50000.WAIT_VAG3:
		M_Activity_WaitingPressure(
			index		:= E_CRYO_EVAC_PRESSURES_50000.VAG3, 
			lrRef		:= cfg.lrThld_Prevac, 
			nNextState	:= E_CRYO_EVAC_STATE_50000.OPEN_PVV1);

	E_CRYO_EVAC_STATE_50000.OPEN_PVV1:
		M_Activity_OpeningValve(
			index		:= E_CRYO_EVAC_VALVES_50000.PVV1, 
			nNextState	:= E_CRYO_EVAC_STATE_50000.WAIT_VAG_1_3);

	E_CRYO_EVAC_STATE_50000.WAIT_VAG_1_3:
		M_Activity_Waiting2Pressures(
			index1		:= E_CRYO_EVAC_PRESSURES_50000.VAG1, 
			index2		:= E_CRYO_EVAC_PRESSURES_50000.VAG3, 
			lrRef		:= cfg.lrThld_Prevac, 
			nNextState	:= E_CRYO_EVAC_STATE_50000.OPEN_PVV2);

	E_CRYO_EVAC_STATE_50000.OPEN_PVV2:
		M_Activity_OpeningValve(
			index		:= E_CRYO_EVAC_VALVES_50000.PVV2, 
			nNextState	:= E_CRYO_EVAC_STATE_50000.WAIT_VAG_F_G_1);

	E_CRYO_EVAC_STATE_50000.WAIT_VAG_F_G_1:
		M_Activity_Waiting2Pressures(
			index1		:= E_CRYO_EVAC_PRESSURES_50000.VAGF, 
			index2		:= E_CRYO_EVAC_PRESSURES_50000.VAGG, 
			lrRef		:= 0.9 * cfg.lrThld_Prevac, 
			nNextState	:= E_CRYO_EVAC_STATE_50000.CLOSE_PVV2);

	E_CRYO_EVAC_STATE_50000.CLOSE_PVV2:
		M_Activity_ClosingValve(
			index		:= E_CRYO_EVAC_VALVES_50000.PVV2, 
			nNextState	:= E_CRYO_EVAC_STATE_50000.CLOSE_PVV1);

	E_CRYO_EVAC_STATE_50000.CLOSE_PVV1:
		M_Activity_ClosingValve(
			index		:= E_CRYO_EVAC_VALVES_50000.PVV1, 
			nNextState	:= E_CRYO_EVAC_STATE_50000.START_TMP);

	E_CRYO_EVAC_STATE_50000.START_TMP:
		M_Activity_StartingTMP();
		
	E_CRYO_EVAC_STATE_50000.OPEN_PVV3:
		M_Activity_OpeningValve(
			index		:= E_CRYO_EVAC_VALVES_50000.PVV3, 
			nNextState	:= E_CRYO_EVAC_STATE_50000.WAIT_VAG_2_3);

	E_CRYO_EVAC_STATE_50000.WAIT_VAG_2_3:
		M_Activity_Waiting2Pressures(
			index1		:= E_CRYO_EVAC_PRESSURES_50000.VAG2, 
			index2		:= E_CRYO_EVAC_PRESSURES_50000.VAG3, 
			lrRef		:= cfg.lrThld_Prevac, 
			nNextState	:= E_CRYO_EVAC_STATE_50000.OPEN_PVV4);

	E_CRYO_EVAC_STATE_50000.OPEN_PVV4:
		M_Activity_OpeningValve(
			index		:= E_CRYO_EVAC_VALVES_50000.PVV4, 
			nNextState	:= E_CRYO_EVAC_STATE_50000.WAIT_VAG_F_G_2);

	E_CRYO_EVAC_STATE_50000.WAIT_VAG_F_G_2:
		M_Activity_Waiting2Pressures(
			index1		:= E_CRYO_EVAC_PRESSURES_50000.VAGF, 
			index2		:= E_CRYO_EVAC_PRESSURES_50000.VAGG, 
			lrRef		:= cfg.lrThld_Vacuum, 
			nNextState	:= E_CRYO_EVAC_STATE_50000.CLOSE_GBV);

	E_CRYO_EVAC_STATE_50000.CLOSE_GBV:
		M_Activity_ClosingValve(
			index		:= E_CRYO_EVAC_VALVES_50000.GBV, 
			nNextState	:= E_CRYO_EVAC_STATE_50000.EVACUATING);

	E_CRYO_EVAC_STATE_50000.EVACUATING:
		M_Activity_Evacuating();

	E_CRYO_EVAC_STATE_50000.CLOSE_ALL_VALVES:
		M_Activity_ClosingAllValves();

	E_CRYO_EVAC_STATE_50000.DELAY_STOPPING:
		M_Activity_DelayBeforeStoppingPumps();

	E_CRYO_EVAC_STATE_50000.STOP_TMP_1:
		M_Activity_StoppingTMP(1);

	E_CRYO_EVAC_STATE_50000.STOP_PVP:
		M_Activity_StoppingPVP();

	E_CRYO_EVAC_STATE_50000.WAIT_TMP_STANDSTILL:
		M_Activity_WaitingTMP2Stop();

	E_CRYO_EVAC_STATE_50000.STOP_TMP_2:
		M_Activity_StoppingTMP(2);

	
END_CASE
END_METHOD

METHOD M_UpdateStatus
VAR_INPUT
END_VAR
stat.bEnabled		:= in_bEnable;
stat.bRootPumpON	:= rpRef.M_IsReady();
stat.bTurboPumpON	:= tpRef.M_IsReady();
END_METHOD

END_FUNCTION_BLOCK

// POUs/Subsystems/Examples/Evacuation/FB_CRYO_EVAC_MICADO
FUNCTION_BLOCK FB_CRYO_EVAC_MICADO EXTENDS FB_CRYO_EVAC_BASE_50000
VAR_INPUT
END_VAR
VAR_OUTPUT
END_VAR
VAR
	// Specify pumps
	rp:	FB_CRYO_PUMP_ECODRY;	// Roughing Pump
	tp:	FB_CRYO_PUMP_ATH2303M;	// Turbomolecular Pump
	
END_VAR

SUPER^();	// Execute base FB code.

METHOD M_Configure
VAR_INPUT
END_VAR
//
// Specific MICADO configuration.
//
IF NOT stat.bConfigured	THEN
	//
	// MANDATORY !!!
	// Call base FB::M_Configure() to set the pointers.
	//
	SUPER^.M_Configure();
	

	// MANDATORY: Set References for pumps!!!
	// If not done, system will crash !!!
	rpRef	REF=rp;
	tpRef	REF=tp;
	

	// Specific instance configuration, e.g. anything different
	// from the default values given in the cfg structure of type T_CRYO_EVAC_CFG_50000.
	cfg.nType_VAG1	:= E_CRYO_SENSOR_TYPE_PRESS.WRG_D_NW25;
	cfg.nType_VAG2	:= E_CRYO_SENSOR_TYPE_PRESS.WRG_D_NW25;
	cfg.nType_VAG3	:= E_CRYO_SENSOR_TYPE_PRESS.WRG_D_NW25;
	cfg.nType_VAGF1	:= E_CRYO_SENSOR_TYPE_PRESS.PKR_250;
	cfg.nType_VAGF2	:= E_CRYO_SENSOR_TYPE_PRESS.PKR_250;
	cfg.nType_VAGG1	:= E_CRYO_SENSOR_TYPE_PRESS.PKR_250;
	cfg.nType_VAGG2	:= E_CRYO_SENSOR_TYPE_PRESS.PKR_250;


	stat.bConfigured	:= TRUE;
ELSE
	RETURN;	// Nothing to do any more
END_IF
END_METHOD

METHOD M_ExecuteControllers
VAR_INPUT
END_VAR
//
// Specific MICADO Evacuation System HW configuration.
//

// Roughing Pump	
rp(	
	in_bSimulation	:= FALSE,
	in_sName		:= 'ECODRY V01',
	in_bEnable		:= ctrl.bEnable_PVP,
	in_nSlaveID		:= 31,
	in_sVersion		:= 'V01',
	in_nPeriod		:= 2000);

// Turbo Molecular Pump
tp(	
	in_bSimulation	:= FALSE,
	in_sName		:= 'ATH2303M',
	in_bEnable		:= ctrl.bEnable_TMP,
	in_nModel		:= 2303,
	in_bAutoMonitor	:= TRUE,
	in_nPeriod		:= 2000);

// Valves are controlled in the base FB
SUPER^.M_ExecuteControllers();
END_METHOD

END_FUNCTION_BLOCK

// POUs/Subsystems/Examples/Evacuation/FB_CRYO_EVAC_ECODRY_ATH2303M
FUNCTION_BLOCK FB_CRYO_EVAC_ECODRY_ATH2303M EXTENDS FB_CRYO_EVAC_BASE
VAR_INPUT
END_VAR
VAR_OUTPUT
END_VAR
VAR
	rp:	FB_CRYO_PUMP_ECODRY;	// Roughing Pump
	tp:	FB_CRYO_PUMP_ATH2303M;	// Turbo Molecular Pump
	
END_VAR

SUPER^();

METHOD M_Configure
VAR_INPUT
END_VAR
//
// Specific PDS IR Imager configuration.
//
IF NOT stat.bConfigured	THEN
	// MANDATORY: Set References !!!
	// If not done, system will crash !!!
	rpRef	REF=rp;
	tpRef	REF=tp;
	

	// Specific instance configuration, e.g. anything different
	// from the default values given in the cfg structure of type T_CRYO_EVAC_CFG.
	cfg.nPressGaugeType1	:= E_CRYO_SENSOR_TYPE_PRESS.WRG_D_NW25;
	cfg.nPressGaugeType2	:= E_CRYO_SENSOR_TYPE_PRESS.PKR_360;

